  MoveL 1900 to (-42.03, -4.8, 85) mm, rotated rx 180 ry 0 rz -180 deg; joints [35.612, 47.892, 27.55, -143.499, 78.209, -188.599]
  Set speed (130.0 mm/s)
  MoveL 1901 to (-54.1, -7.67, 85) mm, rotated rx 180 ry 0 rz -180 deg; joints [36.421, 46.753, 30.307, -142.872, 79.619, -187.768]
  Call Extruder(18350.601)
  Set speed (30.0 mm/s)
  MoveL 1902 to (-53.59, -12.23, 85) mm, rotated rx 180 ry 0 rz -180 deg; joints [35.732, 46.533, 30.847, -143.601, 79.784, -187.449]
  Call Extruder(18361.531)
  MoveL 1903 to (-49.53, -23.85, 85) mm, rotated rx 180 ry 0 rz -180 deg; joints [33.663, 46.219, 31.622, -145.735, 79.903, -186.811]
  Call Extruder(18372.461)
  MoveL 1904 to (-42.98, -34.27, 85) mm, rotated rx 180 ry 0 rz -180 deg; joints [31.506, 46.21, 31.644, -147.914, 79.666, -186.417]
  Call Extruder(18383.391)
  MoveL 1905 to (-34.27, -42.98, 85) mm, rotated rx 180 ry 0 rz -180 deg; joints [29.427, 46.506, 30.913, -149.974, 79.064, -186.258]
  Call Extruder(18394.322)
  MoveL 1906 to (-23.85, -49.52, 85) mm, rotated rx 180 ry 0 rz 180 deg; joints [27.581, 47.095, 29.473, -151.762, 78.118, -186.31]
  Call Extruder(18405.252)
  MoveL 1907 to (-12.23, -53.59, 85) mm, rotated rx 180 ry 0 rz 180 deg; joints [26.087, 47.95, 27.412, -153.159, 76.881, -186.552]
  Call Extruder(18416.182)
  MoveL 1908 to (0, -54.97, 85) mm, rotated rx 180 ry 0 rz -180 deg; joints [25.019, 49.033, 24.845, -154.089, 75.426, -186.97]
  Call Extruder(18421.833)
  MoveL 1909 to (6.32, -54.26, 85) mm, rotated rx -180 ry 0 rz -180 deg; joints [24.697, 49.678, 23.338, -154.319, 74.609, -187.273]
  Call Extruder(18427.112)
  MoveL 1910 to (12.23, -53.59, 85) mm, rotated rx -180 ry 0 rz -180 deg; joints [24.406, 50.294, 21.91, -154.52, 73.84, -187.555]
  Call Extruder(18438.042)
  MoveL 1911 to (23.85, -49.52, 85) mm, rotated rx 180 ry 0 rz 180 deg; joints [24.239, 51.674, 18.756, -154.459, 72.215, -188.304]
  Call Extruder(18448.973)
  MoveL 1912 to (34.27, -42.98, 85) mm, rotated rx 180 ry 0 rz 180 deg; joints [24.487, 53.106, 15.533, -153.939, 70.641, -189.208]
  Call Extruder(18459.903)
  MoveL 1913 to (42.98, -34.27, 85) mm, rotated rx 180 ry 0 rz 180 deg; joints [25.101, 54.522, 12.393, -153.013, 69.203, -190.249]
  Call Extruder(18470.833)
  MoveL 1914 to (49.52, -23.85, 85) mm, rotated rx 180 ry 0 rz -180 deg; joints [26.025, 55.85, 9.486, -151.751, 67.976, -191.391]
  Call Extruder(18481.763)
  MoveL 1915 to (53.59, -12.23, 85) mm, rotated rx -180 ry 0 rz 180 deg; joints [27.2, 57.019, 6.95, -150.232, 67.025, -192.585]
  Call Extruder(18492.693)
  MoveL 1916 to (54.97, 0, 85) mm, rotated rx -180 ry 0 rz -180 deg; joints [28.57, 57.965, 4.914, -148.541, 66.399, -193.763]
  Call Extruder(18503.624)
  MoveL 1917 to (53.59, 12.23, 85) mm, rotated rx 180 ry 0 rz -180 deg; joints [30.077, 58.634, 3.483, -146.767, 66.128, -194.851]
  Call Extruder(18514.554)
  MoveL 1918 to (49.53, 23.85, 85) mm, rotated rx -180 ry 0 rz -180 deg; joints [31.665, 58.984, 2.736, -144.994, 66.219, -195.771]
  Call Extruder(18525.484)
  MoveL 1919 to (42.98, 34.27, 85) mm, rotated rx 180 ry 0 rz 180 deg; joints [33.282, 58.994, 2.714, -143.296, 66.658, -196.456]
  Call Extruder(18536.414)
  MoveL 1920 to (34.27, 42.98, 85) mm, rotated rx 180 ry 0 rz 180 deg; joints [34.874, 58.664, 3.42, -141.736, 67.412, -196.854]
  Call Extruder(18547.344)
  MoveL 1921 to (23.85, 49.53, 85) mm, rotated rx 180 ry 0 rz 180 deg; joints [36.387, 58.013, 4.812, -140.363, 68.428, -196.939]
  Call Extruder(18558.275)
  MoveL 1922 to (12.23, 53.59, 85) mm, rotated rx 180 ry 0 rz -180 deg; joints [37.766, 57.081, 6.816, -139.215, 69.646, -196.703]
  Call Extruder(18569.205)
  MoveL 1923 to (0, 54.97, 85) mm, rotated rx 180 ry 0 rz 180 deg; joints [38.954, 55.923, 9.325, -138.323, 70.999, -196.165]
  Call Extruder(18580.135)
  MoveL 1924 to (-12.23, 53.59, 85) mm, rotated rx 180 ry 0 rz 180 deg; joints [39.895, 54.603, 12.215, -137.717, 72.421, -195.358]
  Call Extruder(18591.065)
  MoveL 1925 to (-23.85, 49.53, 85) mm, rotated rx 180 ry 0 rz 180 deg; joints [40.528, 53.191, 15.344, -137.428, 73.851, -194.333]
  Call Extruder(18601.995)
  MoveL 1926 to (-34.27, 42.98, 85) mm, rotated rx 180 ry 0 rz -180 deg; joints [40.799, 51.757, 18.566, -137.489, 75.233, -193.151]
  Call Extruder(18612.926)
  MoveL 1927 to (-42.98, 34.27, 85) mm, rotated rx -180 ry 0 rz -180 deg; joints [40.659, 50.372, 21.729, -137.932, 76.518, -191.883]
  Call Extruder(18623.856)
  MoveL 1928 to (-49.53, 23.85, 85) mm, rotated rx 180 ry 0 rz 180 deg; joints [40.072, 49.103, 24.681, -138.778, 77.661, -190.604]
  Call Extruder(18634.786)
  MoveL 1929 to (-53.59, 12.23, 85) mm, rotated rx 180 ry 0 rz 180 deg; joints [39.031, 48.008, 27.273, -140.031, 78.617, -189.393]
  Call Extruder(18645.716)
  MoveL 1930 to (-54.97, 0, 85) mm, rotated rx 180 ry 0 rz 180 deg; joints [37.56, 47.138, 29.368, -141.662, 79.34, -188.322]
  Call Extruder(18651.242)
  MoveL 1931 to (-54.27, -6.18, 85) mm, rotated rx 180 ry 0 rz -180 deg; joints [36.644, 46.826, 30.128, -142.636, 79.565, -187.874]
  Set speed (130.0 mm/s)
  MoveL 1932 to (-49.9, -9.51, 85) mm, rotated rx 180 ry 0 rz 180 deg; joints [35.741, 46.98, 29.754, -143.521, 79.265, -187.842]
  MoveL 1933 to (1.69, -13.14, 85) mm, rotated rx -180 ry 0 rz 180 deg; joints [30.694, 51.344, 19.505, -147.855, 73.614, -190.053]
  Call Extruder(18653.246)
  Set speed (80.0 mm/s)
  MoveL 1934 to (2.97, -12.99, 85) mm, rotated rx 180 ry 0 rz -180 deg; joints [30.614, 51.477, 19.201, -147.91, 73.456, -190.124]
  Call Extruder(18657.910)
  MoveL 1935 to (5.78, -12.01, 85) mm, rotated rx 180 ry 0 rz -180 deg; joints [30.526, 51.813, 18.439, -147.933, 73.079, -190.334]
  Call Extruder(18662.573)
  MoveL 1936 to (8.31, -10.42, 85) mm, rotated rx 180 ry 0 rz -180 deg; joints [30.538, 52.16, 17.656, -147.849, 72.712, -190.58]
  Call Extruder(18667.238)
  MoveL 1937 to (10.42, -8.31, 85) mm, rotated rx -180 ry 0 rz -180 deg; joints [30.649, 52.499, 16.893, -147.664, 72.374, -190.852]
  Call Extruder(18671.901)
  MoveL 1938 to (12.01, -5.78, 85) mm, rotated rx 180 ry 0 rz 180 deg; joints [30.85, 52.813, 16.187, -147.389, 72.082, -191.136]
  Call Extruder(18676.565)
  MoveL 1939 to (12.99, -2.97, 85) mm, rotated rx 180 ry 0 rz 180 deg; joints [31.131, 53.088, 15.574, -147.04, 71.852, -191.418]
  Call Extruder(18681.229)
  MoveL 1940 to (13.33, 0, 85) mm, rotated rx 180 ry 0 rz -180 deg; joints [31.476, 53.308, 15.084, -146.635, 71.695, -191.685]
  Call Extruder(18685.893)
  MoveL 1941 to (13, 2.97, 85) mm, rotated rx 180 ry 0 rz -180 deg; joints [31.869, 53.462, 14.741, -146.195, 71.618, -191.923]
  Call Extruder(18690.556)
  MoveL 1942 to (12.01, 5.78, 85) mm, rotated rx -180 ry 0 rz -180 deg; joints [32.292, 53.542, 14.562, -145.741, 71.624, -192.118]
  Call Extruder(18695.220)
  MoveL 1943 to (10.42, 8.31, 85) mm, rotated rx -180 ry 0 rz 180 deg; joints [32.725, 53.544, 14.557, -145.294, 71.713, -192.26]
  Call Extruder(18699.884)
  MoveL 1944 to (8.31, 10.42, 85) mm, rotated rx 180 ry 0 rz 180 deg; joints [33.149, 53.469, 14.725, -144.876, 71.88, -192.341]
  Call Extruder(18704.548)
  MoveL 1945 to (5.78, 12.01, 85) mm, rotated rx 180 ry 0 rz -180 deg; joints [33.544, 53.319, 15.059, -144.504, 72.114, -192.354]
  Call Extruder(18709.211)
  MoveL 1946 to (2.97, 13, 85) mm, rotated rx 180 ry 0 rz 180 deg; joints [33.893, 53.102, 15.541, -144.196, 72.405, -192.301]
  Call Extruder(18713.875)
  MoveL 1947 to (0, 13.33, 85) mm, rotated rx -180 ry 0 rz -180 deg; joints [34.177, 52.831, 16.148, -143.967, 72.737, -192.182]
  Call Extruder(18718.539)
  MoveL 1948 to (-2.97, 13, 85) mm, rotated rx 180 ry 0 rz -180 deg; joints [34.384, 52.518, 16.85, -143.826, 73.094, -192.004]
  Call Extruder(18723.203)
  MoveL 1949 to (-5.78, 12.01, 85) mm, rotated rx 180 ry 0 rz 180 deg; joints [34.5, 52.18, 17.61, -143.782, 73.459, -191.778]
  Call Extruder(18727.866)
  MoveL 1950 to (-8.31, 10.42, 85) mm, rotated rx -180 ry 0 rz -180 deg; joints [34.518, 51.834, 18.393, -143.839, 73.815, -191.515]
  Call Extruder(18732.531)
  MoveL 1951 to (-10.42, 8.31, 85) mm, rotated rx 180 ry 0 rz -180 deg; joints [34.436, 51.496, 19.158, -143.995, 74.144, -191.229]
  Call Extruder(18737.194)
  MoveL 1952 to (-12.01, 5.78, 85) mm, rotated rx -180 ry 0 rz 180 deg; joints [34.254, 51.185, 19.867, -144.246, 74.431, -190.937]
  Call Extruder(18741.858)
  MoveL 1953 to (-12.99, 2.97, 85) mm, rotated rx 180 ry 0 rz -180 deg; joints [33.981, 50.915, 20.484, -144.58, 74.662, -190.654]
  Call Extruder(18746.522)
  MoveL 1954 to (-13.33, 0, 85) mm, rotated rx -180 ry 0 rz -180 deg; joints [33.63, 50.699, 20.978, -144.982, 74.826, -190.393]
  Call Extruder(18751.186)
  MoveL 1955 to (-13, -2.97, 85) mm, rotated rx 180 ry 0 rz 180 deg; joints [33.218, 50.548, 21.325, -145.432, 74.913, -190.167]
  Call Extruder(18755.849)
  MoveL 1956 to (-12.01, -5.78, 85) mm, rotated rx 180 ry 0 rz 180 deg; joints [32.767, 50.47, 21.505, -145.908, 74.918, -189.988]
  Call Extruder(18760.513)
  MoveL 1957 to (-10.42, -8.31, 85) mm, rotated rx -180 ry 0 rz 180 deg; joints [32.302, 50.467, 21.51, -146.382, 74.841, -189.863]
  Call Extruder(18765.177)
  MoveL 1958 to (-8.31, -10.42, 85) mm, rotated rx 180 ry 0 rz -180 deg; joints [31.85, 50.541, 21.34, -146.829, 74.683, -189.797]
  Call Extruder(18769.841)
  MoveL 1959 to (-5.78, -12.01, 85) mm, rotated rx -180 ry 0 rz 180 deg; joints [31.435, 50.688, 21.003, -147.225, 74.453, -189.791]
  Call Extruder(18774.504)
  MoveL 1960 to (-2.97, -12.99, 85) mm, rotated rx 180 ry 0 rz 180 deg; joints [31.079, 50.9, 20.517, -147.548, 74.161, -189.846]
  Call Extruder(18779.168)
  MoveL 1961 to (0, -13.33, 85) mm, rotated rx 180 ry 0 rz -180 deg; joints [30.801, 51.168, 19.906, -147.78, 73.823, -189.959]
  Call Extruder(18781.828)
  MoveL 1962 to (1.69, -13.14, 85) mm, rotated rx -180 ry 0 rz 180 deg; joints [30.694, 51.344, 19.505, -147.855, 73.614, -190.053]
  Set speed (130.0 mm/s)
  MoveL 1963 to (1.69, -13.14, 90) mm, rotated rx -180 ry 0 rz 180 deg; joints [30.694, 50.443, 19.819, -147.761, 73.118, -190.379]
  MoveL 1964 to (-26.25, -4.54, 90) mm, rotated rx 180 ry 0 rz -180 deg; joints [34.172, 48.315, 24.645, -144.623, 75.968, -189.768]
  Call Extruder(18784.060)
  Set speed (60.0 mm/s)
  MoveL 1965 to (-26.09, -5.96, 90) mm, rotated rx 180 ry 0 rz -180 deg; joints [33.969, 48.243, 24.81, -144.843, 76.01, -189.663]
  Call Extruder(18793.425)
  MoveL 1966 to (-24.12, -11.61, 90) mm, rotated rx 180 ry 0 rz 180 deg; joints [33.033, 48.083, 25.176, -145.823, 76.027, -189.311]
  Call Extruder(18802.790)
  MoveL 1967 to (-20.93, -16.69, 90) mm, rotated rx 180 ry 0 rz -180 deg; joints [32.066, 48.079, 25.187, -146.809, 75.877, -189.069]
  Call Extruder(18812.155)
  MoveL 1968 to (-16.69, -20.93, 90) mm, rotated rx 180 ry 0 rz 180 deg; joints [31.126, 48.229, 24.841, -147.739, 75.565, -188.942]
  Call Extruder(18821.520)
  MoveL 1969 to (-11.61, -24.11, 90) mm, rotated rx 180 ry 0 rz -180 deg; joints [30.272, 48.527, 24.158, -148.558, 75.105, -188.931]
  Call Extruder(18830.885)
  MoveL 1970 to (-5.96, -26.09, 90) mm, rotated rx -180 ry 0 rz -180 deg; joints [29.552, 48.958, 23.173, -149.218, 74.519, -189.035]
  Call Extruder(18840.250)
  MoveL 1971 to (0, -26.77, 90) mm, rotated rx -180 ry 0 rz -180 deg; joints [29.003, 49.501, 21.939, -149.681, 73.837, -189.246]
  Call Extruder(18845.916)
  MoveL 1972 to (3.6, -26.36, 90) mm, rotated rx 180 ry 0 rz 180 deg; joints [28.788, 49.881, 21.082, -149.832, 73.389, -189.435]
  Call Extruder(18849.615)
  MoveL 1973 to (5.96, -26.09, 90) mm, rotated rx 180 ry 0 rz 180 deg; joints [28.65, 50.131, 20.519, -149.926, 73.096, -189.558]
  Call Extruder(18858.980)
  MoveL 1974 to (11.61, -24.11, 90) mm, rotated rx 180 ry 0 rz -180 deg; joints [28.503, 50.816, 18.985, -149.946, 72.336, -189.958]
  Call Extruder(18868.345)
  MoveL 1975 to (16.69, -20.93, 90) mm, rotated rx 180 ry 0 rz -180 deg; joints [28.559, 51.523, 17.413, -149.746, 71.598, -190.433]
  Call Extruder(18877.710)
  MoveL 1976 to (20.93, -16.69, 90) mm, rotated rx 180 ry 0 rz 180 deg; joints [28.808, 52.216, 15.882, -149.344, 70.922, -190.964]
  Call Extruder(18887.075)
  MoveL 1977 to (24.12, -11.61, 90) mm, rotated rx -180 ry 0 rz 180 deg; joints [29.229, 52.861, 14.466, -148.767, 70.343, -191.529]
  Call Extruder(18896.440)
  MoveL 1978 to (26.09, -5.96, 90) mm, rotated rx 180 ry 0 rz 180 deg; joints [29.796, 53.424, 13.236, -148.05, 69.891, -192.102]
  Call Extruder(18905.805)
  MoveL 1979 to (26.77, 0, 90) mm, rotated rx 180 ry 0 rz -180 deg; joints [30.482, 53.877, 12.252, -147.232, 69.589, -192.652]
  Call Extruder(18915.170)
  MoveL 1980 to (26.09, 5.96, 90) mm, rotated rx 180 ry 0 rz -180 deg; joints [31.252, 54.194, 11.564, -146.354, 69.451, -193.15]
  Call Extruder(18924.535)
  MoveL 1981 to (24.11, 11.61, 90) mm, rotated rx -180 ry 0 rz 180 deg; joints [32.076, 54.36, 11.205, -145.458, 69.481, -193.565]
  Call Extruder(18933.900)
  MoveL 1982 to (20.93, 16.69, 90) mm, rotated rx 180 ry 0 rz -180 deg; joints [32.917, 54.365, 11.195, -144.584, 69.676, -193.873]
  Call Extruder(18943.265)
  MoveL 1983 to (16.69, 20.93, 90) mm, rotated rx 180 ry 0 rz -180 deg; joints [33.742, 54.208, 11.533, -143.77, 70.023, -194.053]
  Call Extruder(18952.630)
  MoveL 1984 to (11.61, 24.12, 90) mm, rotated rx -180 ry 0 rz 180 deg; joints [34.517, 53.899, 12.203, -143.049, 70.501, -194.094]
  Call Extruder(18961.995)
  MoveL 1985 to (5.96, 26.09, 90) mm, rotated rx 180 ry 0 rz -180 deg; joints [35.208, 53.454, 13.171, -142.449, 71.085, -193.993]
  Call Extruder(18971.360)
  MoveL 1986 to (0, 26.77, 90) mm, rotated rx 180 ry 0 rz 180 deg; joints [35.784, 52.897, 14.388, -141.996, 71.744, -193.754]
  Call Extruder(18980.725)
  MoveL 1987 to (-5.96, 26.09, 90) mm, rotated rx 180 ry 0 rz 180 deg; joints [36.214, 52.256, 15.795, -141.709, 72.448, -193.392]
  Call Extruder(18990.090)
  MoveL 1988 to (-11.61, 24.12, 90) mm, rotated rx 180 ry 0 rz -180 deg; joints [36.473, 51.564, 17.321, -141.605, 73.162, -192.928]
  Call Extruder(18999.455)
  MoveL 1989 to (-16.69, 20.93, 90) mm, rotated rx 180 ry 0 rz -180 deg; joints [36.542, 50.857, 18.893, -141.694, 73.854, -192.389]
  Call Extruder(19008.820)
  MoveL 1990 to (-20.93, 16.69, 90) mm, rotated rx -180 ry 0 rz 180 deg; joints [36.407, 50.17, 20.431, -141.981, 74.495, -191.805]
  Call Extruder(19018.185)
  MoveL 1991 to (-24.12, 11.61, 90) mm, rotated rx -180 ry 0 rz -180 deg; joints [36.065, 49.536, 21.86, -142.46, 75.056, -191.209]
  Call Extruder(19027.550)
  MoveL 1992 to (-26.09, 5.96, 90) mm, rotated rx 180 ry 0 rz -180 deg; joints [35.528, 48.987, 23.107, -143.116, 75.509, -190.634]
  Call Extruder(19036.915)
  MoveL 1993 to (-26.77, 0, 90) mm, rotated rx 180 ry 0 rz -180 deg; joints [34.817, 48.549, 24.108, -143.924, 75.834, -190.11]
  Call Extruder(19041.703)
  MoveL 1994 to (-26.42, -3.05, 90) mm, rotated rx -180 ry 0 rz -180 deg; joints [34.385, 48.391, 24.47, -144.392, 75.924, -189.88]
  Set speed (130.0 mm/s)
  MoveL 1995 to (-41.86, -6.29, 90) mm, rotated rx 180 ry 0 rz -180 deg; joints [35.393, 46.847, 28.05, -143.651, 77.737, -188.884]
  Call Extruder(19046.701)
  Set speed (60.0 mm/s)
  MoveL 1996 to (-41.5, -9.47, 90) mm, rotated rx 180 ry 0 rz 180 deg; joints [34.924, 46.689, 28.423, -144.152, 77.839, -188.654]
  Call Extruder(19061.597)
  MoveL 1997 to (-38.36, -18.47, 90) mm, rotated rx 180 ry 0 rz -180 deg; joints [33.373, 46.437, 29.016, -145.764, 77.892, -188.124]
  Call Extruder(19076.493)
  MoveL 1998 to (-33.29, -26.54, 90) mm, rotated rx 180 ry 0 rz 180 deg; joints [31.763, 46.43, 29.033, -147.397, 77.677, -187.773]
  Call Extruder(19091.389)
  MoveL 1999 to (-26.54, -33.28, 90) mm, rotated rx 180 ry 0 rz -180 deg; joints [30.206, 46.667, 28.474, -148.94, 77.196, -187.603]
  Call Extruder(19106.284)
  MoveL 2000 to (-18.47, -38.36, 90) mm, rotated rx -180 ry 0 rz 180 deg; joints [28.808, 47.137, 27.372, -150.288, 76.465, -187.607]
  Call Extruder(19121.180)
  MoveL 2001 to (-9.47, -41.5, 90) mm, rotated rx 180 ry 0 rz -180 deg; joints [27.654, 47.818, 25.788, -151.357, 75.523, -187.775]
  Call Extruder(19136.076)
  MoveL 2002 to (0, -42.57, 90) mm, rotated rx -180 ry 0 rz -180 deg; joints [26.805, 48.678, 23.811, -152.086, 74.422, -188.098]
  Call Extruder(19144.508)
  MoveL 2003 to (5.36, -41.97, 90) mm, rotated rx 180 ry 0 rz -180 deg; joints [26.51, 49.239, 22.533, -152.294, 73.745, -188.362]
  Call Extruder(19150.972)
  MoveL 2004 to (9.47, -41.5, 90) mm, rotated rx -180 ry 0 rz -180 deg; joints [26.29, 49.676, 21.543, -152.445, 73.223, -188.565]
  Call Extruder(19165.867)
  MoveL 2005 to (18.47, -38.36, 90) mm, rotated rx -180 ry 0 rz -180 deg; joints [26.114, 50.765, 19.1, -152.431, 71.995, -189.168]
  Call Extruder(19180.763)
  MoveL 2006 to (26.54, -33.28, 90) mm, rotated rx 180 ry 0 rz 180 deg; joints [26.262, 51.89, 16.601, -152.062, 70.804, -189.891]
  Call Extruder(19195.659)
  MoveL 2007 to (33.28, -26.54, 90) mm, rotated rx -180 ry 0 rz -180 deg; joints [26.703, 52.997, 14.168, -151.375, 69.715, -190.715]
  Call Extruder(19210.555)
  MoveL 2008 to (38.36, -18.47, 90) mm, rotated rx 180 ry 0 rz 180 deg; joints [27.4, 54.031, 11.918, -150.419, 68.787, -191.607]
  Call Extruder(19225.451)
  MoveL 2009 to (41.5, -9.47, 90) mm, rotated rx 180 ry 0 rz -180 deg; joints [28.309, 54.937, 9.96, -149.255, 68.067, -192.526]
  Call Extruder(19240.347)
  MoveL 2010 to (42.57, 0, 90) mm, rotated rx 180 ry 0 rz 180 deg; joints [29.382, 55.667, 8.391, -147.947, 67.593, -193.424]
  Call Extruder(19255.242)
  MoveL 2011 to (41.5, 9.47, 90) mm, rotated rx 180 ry 0 rz -180 deg; joints [30.575, 56.181, 7.292, -146.562, 67.386, -194.247]
  Call Extruder(19270.138)
  MoveL 2012 to (38.36, 18.47, 90) mm, rotated rx -180 ry 0 rz 180 deg; joints [31.839, 56.449, 6.719, -145.166, 67.452, -194.941]
  Call Extruder(19285.034)
  MoveL 2013 to (33.28, 26.54, 90) mm, rotated rx 180 ry 0 rz -180 deg; joints [33.128, 56.457, 6.702, -143.819, 67.783, -195.459]
  Call Extruder(19299.930)
  MoveL 2014 to (26.54, 33.29, 90) mm, rotated rx 180 ry 0 rz -180 deg; joints [34.394, 56.204, 7.243, -142.573, 68.354, -195.764]
  Call Extruder(19314.826)
  MoveL 2015 to (18.47, 38.36, 90) mm, rotated rx 180 ry 0 rz -180 deg; joints [35.592, 55.703, 8.313, -141.473, 69.129, -195.837]
  Call Extruder(19329.721)
  MoveL 2016 to (9.47, 41.51, 90) mm, rotated rx 180 ry 0 rz -180 deg; joints [36.675, 54.985, 9.856, -140.555, 70.064, -195.67]
  Call Extruder(19344.617)
  MoveL 2017 to (0, 42.57, 90) mm, rotated rx 180 ry 0 rz -180 deg; joints [37.594, 54.088, 11.794, -139.85, 71.109, -195.277]
  Call Extruder(19359.513)
  MoveL 2018 to (-9.47, 41.51, 90) mm, rotated rx 180 ry 0 rz -180 deg; joints [38.304, 53.061, 14.03, -139.386, 72.213, -194.679]
  Call Extruder(19374.409)
  MoveL 2019 to (-18.47, 38.36, 90) mm, rotated rx 180 ry 0 rz -180 deg; joints [38.762, 51.956, 16.455, -139.189, 73.327, -193.915]
  Call Extruder(19389.304)
  MoveL 2020 to (-26.54, 33.29, 90) mm, rotated rx 180 ry 0 rz -180 deg; joints [38.928, 50.83, 18.953, -139.28, 74.405, -193.029]
  Call Extruder(19404.200)
  MoveL 2021 to (-33.29, 26.54, 90) mm, rotated rx 180 ry 0 rz 180 deg; joints [38.772, 49.738, 21.403, -139.676, 75.404, -192.074]
  Call Extruder(19419.096)
  MoveL 2022 to (-38.36, 18.47, 90) mm, rotated rx 180 ry 0 rz 180 deg; joints [38.277, 48.734, 23.684, -140.383, 76.283, -191.106]
  Call Extruder(19433.992)
  MoveL 2023 to (-41.5, 9.47, 90) mm, rotated rx 180 ry 0 rz -180 deg; joints [37.447, 47.864, 25.682, -141.391, 77.005, -190.18]
  Call Extruder(19448.888)
  MoveL 2024 to (-42.57, 0, 90) mm, rotated rx 180 ry 0 rz 180 deg; joints [36.31, 47.172, 27.291, -142.667, 77.535, -189.349]
  Call Extruder(19456.442)
  MoveL 2025 to (-42.03, -4.8, 90) mm, rotated rx -180 ry 0 rz -180 deg; joints [35.612, 46.923, 27.873, -143.416, 77.689, -188.993]
  Set speed (130.0 mm/s)
  MoveL 2026 to (-54.1, -7.67, 90) mm, rotated rx 180 ry 0 rz -180 deg; joints [36.421, 45.756, 30.634, -142.796, 79.086, -188.18]
  Call Extruder(19460.515)
  Set speed (30.0 mm/s)
  MoveL 2027 to (-53.59, -12.23, 90) mm, rotated rx 180 ry 0 rz 180 deg; joints [35.732, 45.53, 31.175, -143.527, 79.242, -187.857]
  Call Extruder(19471.445)
  MoveL 2028 to (-49.53, -23.85, 90) mm, rotated rx 180 ry 0 rz -180 deg; joints [33.663, 45.208, 31.951, -145.665, 79.34, -187.201]
  Call Extruder(19482.375)
  MoveL 2029 to (-42.98, -34.27, 90) mm, rotated rx -180 ry 0 rz -180 deg; joints [31.506, 45.199, 31.974, -147.846, 79.089, -186.786]
  Call Extruder(19493.305)
  MoveL 2030 to (-34.27, -42.98, 90) mm, rotated rx 180 ry 0 rz -180 deg; joints [29.427, 45.503, 31.241, -149.907, 78.479, -186.602]
  Call Extruder(19504.235)
  MoveL 2031 to (-23.85, -49.52, 90) mm, rotated rx 180 ry 0 rz 180 deg; joints [27.581, 46.107, 29.799, -151.694, 77.535, -186.631]
  Call Extruder(19515.166)
  MoveL 2032 to (-12.23, -53.59, 90) mm, rotated rx 180 ry 0 rz 180 deg; joints [26.087, 46.982, 27.734, -153.089, 76.305, -186.852]
  Call Extruder(19526.096)
  MoveL 2033 to (0, -54.97, 90) mm, rotated rx -180 ry 0 rz -180 deg; joints [25.019, 48.089, 25.164, -154.016, 74.864, -187.252]
  Call Extruder(19532.120)
  MoveL 2034 to (6.74, -54.21, 90) mm, rotated rx -180 ry 0 rz 180 deg; joints [24.676, 48.791, 23.554, -154.259, 74.003, -187.569]
  Call Extruder(19537.026)
  MoveL 2035 to (12.23, -53.59, 90) mm, rotated rx 180 ry 0 rz 180 deg; joints [24.406, 49.374, 22.226, -154.444, 73.296, -187.826]
  Call Extruder(19547.956)
  MoveL 2036 to (23.85, -49.53, 90) mm, rotated rx -180 ry 0 rz -180 deg; joints [24.239, 50.778, 19.069, -154.377, 71.691, -188.568]
  Call Extruder(19558.886)
  MoveL 2037 to (34.27, -42.98, 90) mm, rotated rx -180 ry 0 rz 180 deg; joints [24.487, 52.233, 15.845, -153.851, 70.137, -189.47]
  Call Extruder(19569.817)
  MoveL 2038 to (42.98, -34.27, 90) mm, rotated rx -180 ry 0 rz -180 deg; joints [25.101, 53.668, 12.705, -152.918, 68.72, -190.513]
  Call Extruder(19580.747)
  MoveL 2039 to (49.52, -23.85, 90) mm, rotated rx 180 ry 0 rz -180 deg; joints [26.025, 55.012, 9.798, -151.649, 67.514, -191.66]
  Call Extruder(19591.677)
  MoveL 2040 to (53.59, -12.23, 90) mm, rotated rx 180 ry 0 rz 180 deg; joints [27.2, 56.194, 7.264, -150.123, 66.582, -192.862]
  Call Extruder(19602.607)
  MoveL 2041 to (54.97, 0, 90) mm, rotated rx -180 ry 0 rz -180 deg; joints [28.57, 57.15, 5.229, -148.426, 65.973, -194.049]
  Call Extruder(19613.537)
  MoveL 2042 to (53.59, 12.23, 90) mm, rotated rx 180 ry 0 rz 180 deg; joints [30.077, 57.824, 3.799, -146.646, 65.715, -195.147]
  Call Extruder(19624.468)
  MoveL 2043 to (49.52, 23.85, 90) mm, rotated rx 180 ry 0 rz 180 deg; joints [31.665, 58.178, 3.053, -144.869, 65.818, -196.079]
  Call Extruder(19635.398)
  MoveL 2044 to (42.98, 34.27, 90) mm, rotated rx 180 ry 0 rz -180 deg; joints [33.282, 58.188, 3.031, -143.169, 66.266, -196.775]
  Call Extruder(19646.328)
  MoveL 2045 to (34.27, 42.98, 90) mm, rotated rx 180 ry 0 rz 180 deg; joints [34.874, 57.854, 3.736, -141.608, 67.025, -197.186]
  Call Extruder(19657.258)
  MoveL 2046 to (23.85, 49.53, 90) mm, rotated rx 180 ry 0 rz -180 deg; joints [36.387, 57.198, 5.127, -140.236, 68.043, -197.282]
  Call Extruder(19668.188)
  MoveL 2047 to (12.23, 53.59, 90) mm, rotated rx -180 ry 0 rz 180 deg; joints [37.766, 56.257, 7.129, -139.09, 69.26, -197.06]
  Call Extruder(19679.119)
  MoveL 2048 to (0, 54.97, 90) mm, rotated rx -180 ry 0 rz -180 deg; joints [38.954, 55.086, 9.638, -138.201, 70.608, -196.534]
  Call Extruder(19690.049)
  MoveL 2049 to (-12.23, 53.59, 90) mm, rotated rx 180 ry 0 rz 180 deg; joints [39.895, 53.75, 12.527, -137.6, 72.021, -195.741]
  Call Extruder(19700.979)
  MoveL 2050 to (-23.85, 49.53, 90) mm, rotated rx 180 ry 0 rz -180 deg; joints [40.528, 52.319, 15.656, -137.316, 73.439, -194.728]
  Call Extruder(19711.909)
  MoveL 2051 to (-34.27, 42.98, 90) mm, rotated rx -180 ry 0 rz 180 deg; joints [40.799, 50.863, 18.88, -137.384, 74.805, -193.558]
  Call Extruder(19722.839)
  MoveL 2052 to (-42.98, 34.27, 90) mm, rotated rx 180 ry 0 rz -180 deg; joints [40.659, 49.454, 22.045, -137.833, 76.071, -192.299]
  Call Extruder(19733.770)
  MoveL 2053 to (-49.53, 23.85, 90) mm, rotated rx 180 ry 0 rz 180 deg; joints [40.072, 48.16, 25, -138.686, 77.192, -191.026]
  Call Extruder(19744.700)
  MoveL 2054 to (-53.59, 12.23, 90) mm, rotated rx -180 ry 0 rz -180 deg; joints [39.031, 47.042, 27.595, -139.946, 78.123, -189.816]
  Call Extruder(19755.630)
  MoveL 2055 to (-54.97, 0, 90) mm, rotated rx 180 ry 0 rz -180 deg; joints [37.56, 46.151, 29.693, -141.583, 78.822, -188.741]
  Call Extruder(19761.156)
  MoveL 2056 to (-54.27, -6.18, 90) mm, rotated rx 180 ry 0 rz -180 deg; joints [36.644, 45.831, 30.455, -142.559, 79.034, -188.287]
  Set speed (130.0 mm/s)
  MoveL 2057 to (-49.9, -9.51, 90) mm, rotated rx 180 ry 0 rz -180 deg; joints [35.741, 45.989, 30.08, -143.444, 78.731, -188.245]
  MoveL 2058 to (2.11, -13.09, 90) mm, rotated rx 180 ry 0 rz 180 deg; joints [30.668, 50.487, 19.719, -147.779, 73.066, -190.402]
  Call Extruder(19762.504)
  Set speed (80.0 mm/s)
  MoveL 2059 to (2.97, -12.99, 90) mm, rotated rx 180 ry 0 rz 180 deg; joints [30.614, 50.579, 19.515, -147.816, 72.961, -190.449]
  Call Extruder(19767.168)
  MoveL 2060 to (5.78, -12.01, 90) mm, rotated rx -180 ry 0 rz 180 deg; joints [30.526, 50.92, 18.752, -147.838, 72.588, -190.657]
  Call Extruder(19771.831)
  MoveL 2061 to (8.31, -10.42, 90) mm, rotated rx -180 ry 0 rz 180 deg; joints [30.538, 51.272, 17.969, -147.752, 72.226, -190.901]
  Call Extruder(19776.495)
  MoveL 2062 to (10.42, -8.31, 90) mm, rotated rx 180 ry 0 rz -180 deg; joints [30.649, 51.616, 17.206, -147.565, 71.893, -191.172]
  Call Extruder(19781.159)
  MoveL 2063 to (12.01, -5.78, 90) mm, rotated rx 180 ry 0 rz -180 deg; joints [30.85, 51.936, 16.5, -147.289, 71.606, -191.457]
  Call Extruder(19785.823)
  MoveL 2064 to (12.99, -2.97, 90) mm, rotated rx 180 ry 0 rz -180 deg; joints [31.131, 52.214, 15.886, -146.938, 71.381, -191.74]
  Call Extruder(19790.487)
  MoveL 2065 to (13.33, 0, 90) mm, rotated rx 180 ry 0 rz -180 deg; joints [31.476, 52.437, 15.396, -146.532, 71.229, -192.01]
  Call Extruder(19795.150)
  MoveL 2066 to (12.99, 2.97, 90) mm, rotated rx -180 ry 0 rz -180 deg; joints [31.869, 52.593, 15.053, -146.091, 71.156, -192.25]
  Call Extruder(19799.814)
  MoveL 2067 to (12.01, 5.78, 90) mm, rotated rx 180 ry 0 rz -180 deg; joints [32.292, 52.675, 14.874, -145.636, 71.166, -192.448]
  Call Extruder(19804.478)
  MoveL 2068 to (10.42, 8.31, 90) mm, rotated rx 180 ry 0 rz 180 deg; joints [32.725, 52.677, 14.869, -145.188, 71.258, -192.594]
  Call Extruder(19809.142)
  MoveL 2069 to (8.31, 10.42, 90) mm, rotated rx 180 ry 0 rz 180 deg; joints [33.149, 52.6, 15.038, -144.77, 71.425, -192.678]
  Call Extruder(19813.805)
  MoveL 2070 to (5.78, 12.01, 90) mm, rotated rx 180 ry 0 rz 180 deg; joints [33.544, 52.448, 15.371, -144.398, 71.66, -192.696]
  Call Extruder(19818.469)
  MoveL 2071 to (2.97, 13, 90) mm, rotated rx 180 ry 0 rz 180 deg; joints [33.893, 52.229, 15.854, -144.091, 71.95, -192.646]
  Call Extruder(19823.133)
  MoveL 2072 to (0, 13.33, 90) mm, rotated rx 180 ry 0 rz 180 deg; joints [34.177, 51.953, 16.461, -143.862, 72.28, -192.53]
  Call Extruder(19827.797)
  MoveL 2073 to (-2.97, 13, 90) mm, rotated rx 180 ry 0 rz 180 deg; joints [34.384, 51.636, 17.162, -143.722, 72.635, -192.356]
  Call Extruder(19832.461)
  MoveL 2074 to (-5.78, 12.01, 90) mm, rotated rx 180 ry 0 rz 180 deg; joints [34.5, 51.293, 17.923, -143.68, 72.996, -192.132]
  Call Extruder(19837.124)
  MoveL 2075 to (-8.31, 10.42, 90) mm, rotated rx 180 ry 0 rz 180 deg; joints [34.518, 50.941, 18.706, -143.738, 73.347, -191.871]
  Call Extruder(19841.788)
  MoveL 2076 to (-10.42, 8.31, 90) mm, rotated rx -180 ry 0 rz -180 deg; joints [34.436, 50.598, 19.471, -143.896, 73.672, -191.587]
  Call Extruder(19846.452)
  MoveL 2077 to (-12.01, 5.78, 90) mm, rotated rx 180 ry 0 rz 180 deg; joints [34.254, 50.281, 20.181, -144.148, 73.953, -191.296]
  Call Extruder(19851.116)
  MoveL 2078 to (-12.99, 2.97, 90) mm, rotated rx 180 ry 0 rz 180 deg; joints [33.981, 50.006, 20.799, -144.484, 74.179, -191.011]
  Call Extruder(19855.780)
  MoveL 2079 to (-13.33, 0, 90) mm, rotated rx 180 ry 0 rz 180 deg; joints [33.63, 49.787, 21.294, -144.888, 74.337, -190.748]
  Call Extruder(19860.443)
  MoveL 2080 to (-13, -2.97, 90) mm, rotated rx 180 ry 0 rz -180 deg; joints [33.218, 49.633, 21.64, -145.339, 74.42, -190.521]
  Call Extruder(19865.107)
  MoveL 2081 to (-12.01, -5.78, 90) mm, rotated rx 180 ry 0 rz 180 deg; joints [32.767, 49.554, 21.821, -145.815, 74.421, -190.338]
  Call Extruder(19869.771)
  MoveL 2082 to (-10.42, -8.31, 90) mm, rotated rx -180 ry 0 rz -180 deg; joints [32.302, 49.551, 21.826, -146.29, 74.341, -190.208]
  Call Extruder(19874.435)
  MoveL 2083 to (-8.31, -10.42, 90) mm, rotated rx 180 ry 0 rz 180 deg; joints [31.85, 49.627, 21.656, -146.738, 74.182, -190.137]
  Call Extruder(19879.098)
  MoveL 2084 to (-5.78, -12.01, 90) mm, rotated rx 180 ry 0 rz -180 deg; joints [31.435, 49.776, 21.318, -147.134, 73.951, -190.127]
  Call Extruder(19883.762)
  MoveL 2085 to (-2.97, -12.99, 90) mm, rotated rx 180 ry 0 rz 180 deg; joints [31.079, 49.992, 20.832, -147.456, 73.661, -190.178]
  Call Extruder(19888.426)
  MoveL 2086 to (0, -13.33, 90) mm, rotated rx 180 ry 0 rz 180 deg; joints [30.801, 50.264, 20.22, -147.687, 73.325, -190.287]
  Call Extruder(19891.742)
  MoveL 2087 to (2.11, -13.09, 90) mm, rotated rx 180 ry 0 rz 180 deg; joints [30.668, 50.487, 19.719, -147.779, 73.066, -190.402]
  Set speed (130.0 mm/s)
  MoveL 2088 to (2.11, -13.09, 95) mm, rotated rx 180 ry 0 rz -180 deg; joints [30.668, 49.592, 20.016, -147.681, 72.561, -190.736]
  MoveL 2089 to (-26.25, -4.54, 95) mm, rotated rx 180 ry 0 rz -180 deg; joints [34.172, 47.38, 24.946, -144.529, 75.452, -190.147]
  Call Extruder(19893.974)
  Set speed (60.0 mm/s)
  MoveL 2090 to (-26.09, -5.96, 95) mm, rotated rx 180 ry 0 rz 180 deg; joints [33.969, 47.306, 25.111, -144.75, 75.492, -190.04]
  Call Extruder(19903.339)
  MoveL 2091 to (-24.12, -11.61, 95) mm, rotated rx -180 ry 0 rz 180 deg; joints [33.033, 47.144, 25.478, -145.732, 75.499, -189.681]
  Call Extruder(19912.704)
  MoveL 2092 to (-20.93, -16.69, 95) mm, rotated rx 180 ry 0 rz -180 deg; joints [32.066, 47.139, 25.489, -146.719, 75.344, -189.43]
  Call Extruder(19922.069)
  MoveL 2093 to (-16.69, -20.93, 95) mm, rotated rx 180 ry 0 rz 180 deg; joints [31.126, 47.293, 25.143, -147.65, 75.029, -189.293]
  Call Extruder(19931.434)
  MoveL 2094 to (-11.61, -24.11, 95) mm, rotated rx 180 ry 0 rz 180 deg; joints [30.272, 47.596, 24.459, -148.469, 74.568, -189.272]
  Call Extruder(19940.799)
  MoveL 2095 to (-5.96, -26.09, 95) mm, rotated rx 180 ry 0 rz -180 deg; joints [29.552, 48.036, 23.473, -149.128, 73.984, -189.366]
  Call Extruder(19950.164)
  MoveL 2096 to (0, -26.77, 95) mm, rotated rx 180 ry 0 rz -180 deg; joints [29.003, 48.589, 22.238, -149.59, 73.307, -189.569]
  Call Extruder(19956.486)
  MoveL 2097 to (4.02, -26.31, 95) mm, rotated rx 180 ry 0 rz -180 deg; joints [28.764, 49.02, 21.28, -149.756, 72.813, -189.775]
  Call Extruder(19959.529)
  MoveL 2098 to (5.96, -26.09, 95) mm, rotated rx 180 ry 0 rz 180 deg; joints [28.65, 49.23, 20.816, -149.833, 72.574, -189.874]
  Call Extruder(19968.894)
  MoveL 2099 to (11.61, -24.11, 95) mm, rotated rx 180 ry 0 rz 180 deg; joints [28.503, 49.927, 19.281, -149.85, 71.823, -190.27]
  Call Extruder(19978.259)
  MoveL 2100 to (16.69, -20.93, 95) mm, rotated rx 180 ry 0 rz -180 deg; joints [28.559, 50.645, 17.709, -149.647, 71.095, -190.743]
  Call Extruder(19987.624)
  MoveL 2101 to (20.93, -16.69, 95) mm, rotated rx 180 ry 0 rz 180 deg; joints [28.808, 51.348, 16.177, -149.242, 70.43, -191.274]
  Call Extruder(19996.989)
  MoveL 2102 to (24.12, -11.61, 95) mm, rotated rx 180 ry 0 rz 180 deg; joints [29.229, 52.002, 14.761, -148.661, 69.861, -191.841]
  Call Extruder(20006.354)
  MoveL 2103 to (26.09, -5.96, 95) mm, rotated rx 180 ry 0 rz 180 deg; joints [29.796, 52.573, 13.531, -147.941, 69.42, -192.416]
  Call Extruder(20015.719)
  MoveL 2104 to (26.77, 0, 95) mm, rotated rx 180 ry 0 rz 180 deg; joints [30.482, 53.031, 12.547, -147.119, 69.127, -192.971]
  Call Extruder(20025.084)
  MoveL 2105 to (26.09, 5.96, 95) mm, rotated rx 180 ry 0 rz 180 deg; joints [31.252, 53.353, 11.859, -146.239, 68.996, -193.474]
  Call Extruder(20034.449)
  MoveL 2106 to (24.11, 11.61, 95) mm, rotated rx 180 ry 0 rz -180 deg; joints [32.076, 53.521, 11.5, -145.341, 69.033, -193.896]
  Call Extruder(20043.814)
  MoveL 2107 to (20.93, 16.69, 95) mm, rotated rx 180 ry 0 rz -180 deg; joints [32.917, 53.525, 11.49, -144.466, 69.233, -194.21]
  Call Extruder(20053.179)
  MoveL 2108 to (16.69, 20.93, 95) mm, rotated rx 180 ry 0 rz 180 deg; joints [33.742, 53.367, 11.828, -143.651, 69.583, -194.398]
  Call Extruder(20062.544)
  MoveL 2109 to (11.61, 24.12, 95) mm, rotated rx -180 ry 0 rz -180 deg; joints [34.517, 53.054, 12.498, -142.93, 70.062, -194.446]
  Call Extruder(20071.908)
  MoveL 2110 to (5.96, 26.09, 95) mm, rotated rx -180 ry 0 rz -180 deg; joints [35.208, 52.603, 13.466, -142.332, 70.645, -194.352]
  Call Extruder(20081.274)
  MoveL 2111 to (0, 26.77, 95) mm, rotated rx 180 ry 0 rz 180 deg; joints [35.784, 52.038, 14.683, -141.88, 71.301, -194.12]
  Call Extruder(20090.639)
  MoveL 2112 to (-5.96, 26.09, 95) mm, rotated rx 180 ry 0 rz -180 deg; joints [36.214, 51.388, 16.09, -141.595, 71.999, -193.765]
  Call Extruder(20100.003)
  MoveL 2113 to (-11.61, 24.12, 95) mm, rotated rx 180 ry 0 rz -180 deg; joints [36.473, 50.687, 17.617, -141.494, 72.706, -193.307]
  Call Extruder(20109.368)
  MoveL 2114 to (-16.69, 20.93, 95) mm, rotated rx 180 ry 0 rz -180 deg; joints [36.542, 49.969, 19.189, -141.586, 73.39, -192.772]
  Call Extruder(20118.734)
  MoveL 2115 to (-20.93, 16.69, 95) mm, rotated rx 180 ry 0 rz 180 deg; joints [36.407, 49.27, 20.729, -141.876, 74.021, -192.191]
  Call Extruder(20128.099)
  MoveL 2116 to (-24.12, 11.61, 95) mm, rotated rx 180 ry 0 rz 180 deg; joints [36.065, 48.625, 22.159, -142.358, 74.57, -191.596]
  Call Extruder(20137.463)
  MoveL 2117 to (-26.09, 5.96, 95) mm, rotated rx 180 ry 0 rz 180 deg; joints [35.528, 48.065, 23.407, -143.018, 75.012, -191.02]
  Call Extruder(20146.828)
  MoveL 2118 to (-26.77, 0, 95) mm, rotated rx 180 ry 0 rz -180 deg; joints [34.817, 47.619, 24.409, -143.828, 75.326, -190.493]
  Call Extruder(20151.617)
  MoveL 2119 to (-26.42, -3.05, 95) mm, rotated rx 180 ry 0 rz -180 deg; joints [34.385, 47.458, 24.771, -144.298, 75.411, -190.26]
  Set speed (130.0 mm/s)
  MoveL 2120 to (-41.86, -6.29, 95) mm, rotated rx 180 ry 0 rz 180 deg; joints [35.393, 45.881, 28.356, -143.564, 77.205, -189.285]
  Call Extruder(20156.615)
  Set speed (60.0 mm/s)
  MoveL 2121 to (-41.5, -9.47, 95) mm, rotated rx -180 ry 0 rz 180 deg; joints [34.924, 45.719, 28.73, -144.067, 77.301, -189.052]
  Call Extruder(20171.511)
  MoveL 2122 to (-38.36, -18.47, 95) mm, rotated rx 180 ry 0 rz 180 deg; joints [33.373, 45.462, 29.323, -145.681, 77.339, -188.509]
  Call Extruder(20186.407)
  MoveL 2123 to (-33.28, -26.54, 95) mm, rotated rx 180 ry 0 rz -180 deg; joints [31.763, 45.454, 29.34, -147.316, 77.114, -188.143]
  Call Extruder(20201.302)
  MoveL 2124 to (-26.54, -33.29, 95) mm, rotated rx -180 ry 0 rz -180 deg; joints [30.206, 45.697, 28.78, -148.86, 76.627, -187.955]
  Call Extruder(20216.198)
  MoveL 2125 to (-18.47, -38.36, 95) mm, rotated rx 180 ry 0 rz 180 deg; joints [28.808, 46.178, 27.676, -150.209, 75.897, -187.942]
  Call Extruder(20231.094)
  MoveL 2126 to (-9.47, -41.5, 95) mm, rotated rx -180 ry 0 rz -180 deg; joints [27.654, 46.874, 26.091, -151.276, 74.96, -188.094]
  Call Extruder(20245.990)
  MoveL 2127 to (0, -42.57, 95) mm, rotated rx -180 ry 0 rz -180 deg; joints [26.805, 47.751, 24.111, -152.002, 73.868, -188.403]
  Call Extruder(20255.078)
  MoveL 2128 to (5.78, -41.92, 95) mm, rotated rx 180 ry 0 rz 180 deg; joints [26.488, 48.367, 22.732, -152.224, 73.146, -188.682]
  Call Extruder(20260.886)
  MoveL 2129 to (9.47, -41.5, 95) mm, rotated rx 180 ry 0 rz -180 deg; joints [26.29, 48.768, 21.841, -152.358, 72.682, -188.861]
  Call Extruder(20275.781)
  MoveL 2130 to (18.47, -38.36, 95) mm, rotated rx 180 ry 0 rz 180 deg; joints [26.114, 49.874, 19.396, -152.34, 71.469, -189.458]
  Call Extruder(20290.677)
  MoveL 2131 to (26.54, -33.28, 95) mm, rotated rx 180 ry 0 rz 180 deg; joints [26.262, 51.017, 16.897, -151.966, 70.294, -190.179]
  Call Extruder(20305.573)
  MoveL 2132 to (33.28, -26.54, 95) mm, rotated rx 180 ry 0 rz 180 deg; joints [26.703, 52.14, 14.463, -151.274, 69.223, -191.003]
  Call Extruder(20320.469)
  MoveL 2133 to (38.36, -18.47, 95) mm, rotated rx -180 ry 0 rz -180 deg; joints [27.4, 53.187, 12.213, -150.313, 68.311, -191.898]
  Call Extruder(20335.364)
  MoveL 2134 to (41.51, -9.47, 95) mm, rotated rx 180 ry 0 rz 180 deg; joints [28.309, 54.104, 10.255, -149.143, 67.606, -192.823]
  Call Extruder(20350.260)
  MoveL 2135 to (42.57, 0, 95) mm, rotated rx 180 ry 0 rz 180 deg; joints [29.382, 54.843, 8.687, -147.83, 67.145, -193.729]
  Call Extruder(20365.156)
  MoveL 2136 to (41.51, 9.47, 95) mm, rotated rx 180 ry 0 rz 180 deg; joints [30.575, 55.362, 7.588, -146.441, 66.95, -194.56]
  Call Extruder(20380.052)
  MoveL 2137 to (38.36, 18.47, 95) mm, rotated rx 180 ry 0 rz -180 deg; joints [31.839, 55.634, 7.015, -145.042, 67.026, -195.263]
  Call Extruder(20394.948)
  MoveL 2138 to (33.28, 26.54, 95) mm, rotated rx 180 ry 0 rz 180 deg; joints [33.128, 55.641, 6.999, -143.692, 67.364, -195.791]
  Call Extruder(20409.843)
  MoveL 2139 to (26.54, 33.29, 95) mm, rotated rx 180 ry 0 rz 180 deg; joints [34.394, 55.385, 7.539, -142.446, 67.939, -196.107]
  Call Extruder(20424.739)
  MoveL 2140 to (18.47, 38.36, 95) mm, rotated rx 180 ry 0 rz -180 deg; joints [35.592, 54.88, 8.609, -141.346, 68.716, -196.19]
  Call Extruder(20439.635)
  MoveL 2141 to (9.47, 41.51, 95) mm, rotated rx 180 ry 0 rz 180 deg; joints [36.675, 54.153, 10.151, -140.429, 69.65, -196.034]
  Call Extruder(20454.531)
  MoveL 2142 to (0, 42.57, 95) mm, rotated rx 180 ry 0 rz -180 deg; joints [37.594, 53.245, 12.089, -139.727, 70.69, -195.651]
  Call Extruder(20469.427)
  MoveL 2143 to (-9.47, 41.5, 95) mm, rotated rx -180 ry 0 rz 180 deg; joints [38.304, 52.205, 14.325, -139.267, 71.788, -195.064]
  Call Extruder(20484.322)
  MoveL 2144 to (-18.47, 38.36, 95) mm, rotated rx 180 ry 0 rz 180 deg; joints [38.762, 51.085, 16.751, -139.074, 72.892, -194.309]
  Call Extruder(20499.218)
  MoveL 2145 to (-26.54, 33.29, 95) mm, rotated rx 180 ry 0 rz 180 deg; joints [38.928, 49.941, 19.249, -139.17, 73.956, -193.431]
  Call Extruder(20514.114)
  MoveL 2146 to (-33.29, 26.54, 95) mm, rotated rx 180 ry 0 rz 180 deg; joints [38.772, 48.831, 21.701, -139.571, 74.939, -192.482]
  Call Extruder(20529.010)
  MoveL 2147 to (-38.36, 18.47, 95) mm, rotated rx 180 ry 0 rz 180 deg; joints [38.277, 47.807, 23.984, -140.283, 75.801, -191.517]
  Call Extruder(20543.906)
  MoveL 2148 to (-41.51, 9.47, 95) mm, rotated rx 180 ry 0 rz 180 deg; joints [37.447, 46.921, 25.984, -141.296, 76.504, -190.592]
  Call Extruder(20558.801)
  MoveL 2149 to (-42.57, 0, 95) mm, rotated rx 180 ry 0 rz -180 deg; joints [36.31, 46.213, 27.596, -142.577, 77.015, -189.756]
  Call Extruder(20566.356)
  MoveL 2150 to (-42.03, -4.8, 95) mm, rotated rx 180 ry 0 rz 180 deg; joints [35.612, 45.959, 28.178, -143.329, 77.16, -189.395]
  Set speed (130.0 mm/s)
  MoveL 2151 to (-54.1, -7.67, 95) mm, rotated rx 180 ry 0 rz 180 deg; joints [36.421, 44.764, 30.944, -142.714, 78.542, -188.601]
  Call Extruder(20570.428)
  Set speed (30.0 mm/s)
  MoveL 2152 to (-53.59, -12.23, 95) mm, rotated rx 180 ry 0 rz -180 deg; joints [35.732, 44.532, 31.486, -143.447, 78.689, -188.274]
  Call Extruder(20581.358)
  MoveL 2153 to (-49.53, -23.85, 95) mm, rotated rx -180 ry 0 rz -180 deg; joints [33.663, 44.201, 32.263, -145.589, 78.767, -187.601]
  Call Extruder(20592.289)
  MoveL 2154 to (-42.98, -34.27, 95) mm, rotated rx 180 ry 0 rz -180 deg; joints [31.506, 44.192, 32.286, -147.772, 78.5, -187.163]
  Call Extruder(20603.219)
  MoveL 2155 to (-34.27, -42.98, 95) mm, rotated rx -180 ry 0 rz -180 deg; joints [29.427, 44.504, 31.552, -149.834, 77.884, -186.955]
  Call Extruder(20614.149)
  MoveL 2156 to (-23.85, -49.53, 95) mm, rotated rx 180 ry 0 rz 180 deg; joints [27.581, 45.123, 30.107, -151.622, 76.94, -186.96]
  Call Extruder(20625.079)
  MoveL 2157 to (-12.23, -53.59, 95) mm, rotated rx -180 ry 0 rz -180 deg; joints [26.087, 46.019, 28.039, -153.015, 75.719, -187.159]
  Call Extruder(20636.010)
  MoveL 2158 to (0, -54.97, 95) mm, rotated rx -180 ry 0 rz 180 deg; joints [25.019, 47.15, 25.466, -153.939, 74.291, -187.543]
  Call Extruder(20642.407)
  MoveL 2159 to (7.16, -54.16, 95) mm, rotated rx 180 ry 0 rz 180 deg; joints [24.655, 47.91, 23.754, -154.194, 73.387, -187.871]
  Call Extruder(20646.940)
  MoveL 2160 to (12.23, -53.59, 95) mm, rotated rx 180 ry 0 rz -180 deg; joints [24.406, 48.46, 22.525, -154.363, 72.741, -188.104]
  Call Extruder(20657.870)
  MoveL 2161 to (23.85, -49.53, 95) mm, rotated rx -180 ry 0 rz -180 deg; joints [24.239, 49.888, 19.366, -154.291, 71.156, -188.839]
  Call Extruder(20668.800)
  MoveL 2162 to (34.27, -42.98, 95) mm, rotated rx 180 ry 0 rz -180 deg; joints [24.487, 51.365, 16.14, -153.758, 69.624, -189.739]
  Call Extruder(20679.730)
  MoveL 2163 to (42.98, -34.27, 95) mm, rotated rx -180 ry 0 rz 180 deg; joints [25.101, 52.82, 13, -152.819, 68.228, -190.784]
  Call Extruder(20690.661)
  MoveL 2164 to (49.52, -23.85, 95) mm, rotated rx 180 ry 0 rz -180 deg; joints [26.025, 54.18, 10.094, -151.543, 67.042, -191.937]
  Call Extruder(20701.591)
  MoveL 2165 to (53.59, -12.23, 95) mm, rotated rx -180 ry 0 rz 180 deg; joints [27.2, 55.375, 7.561, -150.009, 66.129, -193.146]
  Call Extruder(20712.521)
  MoveL 2166 to (54.97, 0, 95) mm, rotated rx -180 ry 0 rz 180 deg; joints [28.57, 56.341, 5.527, -148.305, 65.537, -194.343]
  Call Extruder(20723.451)
  MoveL 2167 to (53.59, 12.23, 95) mm, rotated rx -180 ry 0 rz -180 deg; joints [30.077, 57.022, 4.098, -146.52, 65.295, -195.452]
  Call Extruder(20734.381)
  MoveL 2168 to (49.52, 23.85, 95) mm, rotated rx 180 ry 0 rz 180 deg; joints [31.665, 57.379, 3.352, -144.738, 65.409, -196.395]
  Call Extruder(20745.312)
  MoveL 2169 to (42.98, 34.27, 95) mm, rotated rx 180 ry 0 rz -180 deg; joints [33.282, 57.389, 3.331, -143.035, 65.866, -197.103]
  Call Extruder(20756.242)
  MoveL 2170 to (34.27, 42.98, 95) mm, rotated rx 180 ry 0 rz 180 deg; joints [34.874, 57.052, 4.035, -141.474, 66.631, -197.527]
  Call Extruder(20767.172)
  MoveL 2171 to (23.85, 49.53, 95) mm, rotated rx 180 ry 0 rz -180 deg; joints [36.387, 56.389, 5.425, -140.103, 67.651, -197.636]
  Call Extruder(20778.102)
  MoveL 2172 to (12.23, 53.59, 95) mm, rotated rx 180 ry 0 rz -180 deg; joints [37.766, 55.439, 7.426, -138.959, 68.866, -197.426]
  Call Extruder(20789.032)
  MoveL 2173 to (0, 54.97, 95) mm, rotated rx -180 ry 0 rz -180 deg; joints [38.954, 54.256, 9.933, -138.074, 70.209, -196.913]
  Call Extruder(20799.963)
  MoveL 2174 to (-12.23, 53.59, 95) mm, rotated rx 180 ry 0 rz -180 deg; joints [39.895, 52.903, 12.822, -137.477, 71.614, -196.133]
  Call Extruder(20810.893)
  MoveL 2175 to (-23.85, 49.53, 95) mm, rotated rx -180 ry 0 rz -180 deg; joints [40.528, 51.452, 15.952, -137.2, 73.019, -195.133]
  Call Extruder(20821.823)
  MoveL 2176 to (-34.27, 42.98, 95) mm, rotated rx 180 ry 0 rz 180 deg; joints [40.799, 49.974, 19.176, -137.273, 74.37, -193.974]
  Call Extruder(20832.753)
  MoveL 2177 to (-42.98, 34.27, 95) mm, rotated rx -180 ry 0 rz -180 deg; joints [40.659, 48.542, 22.344, -137.729, 75.616, -192.724]
  Call Extruder(20843.683)
  MoveL 2178 to (-49.52, 23.85, 95) mm, rotated rx -180 ry 0 rz -180 deg; joints [40.072, 47.222, 25.302, -138.589, 76.714, -191.458]
  Call Extruder(20854.614)
  MoveL 2179 to (-53.59, 12.23, 95) mm, rotated rx 180 ry 0 rz 180 deg; joints [39.031, 46.08, 27.9, -139.855, 77.621, -190.249]
  Call Extruder(20865.544)
  MoveL 2180 to (-54.97, 0, 95) mm, rotated rx -180 ry 0 rz 180 deg; joints [37.56, 45.168, 30.002, -141.498, 78.294, -189.169]
  Call Extruder(20871.069)
  MoveL 2181 to (-54.27, -6.18, 95) mm, rotated rx 180 ry 0 rz 180 deg; joints [36.644, 44.841, 30.764, -142.476, 78.494, -188.71]
  Set speed (130.0 mm/s)
  MoveL 2182 to (-49.9, -9.51, 95) mm, rotated rx 180 ry 0 rz -180 deg; joints [35.741, 45.002, 30.389, -143.361, 78.187, -188.657]
  MoveL 2183 to (2.53, -13.04, 95) mm, rotated rx 180 ry 0 rz -180 deg; joints [30.642, 49.638, 19.917, -147.699, 72.51, -190.758]
  Call Extruder(20871.762)
  Set speed (80.0 mm/s)
  MoveL 2184 to (2.97, -12.99, 95) mm, rotated rx -180 ry 0 rz 180 deg; joints [30.614, 49.685, 19.812, -147.717, 72.456, -190.782]
  Call Extruder(20876.425)
  MoveL 2185 to (5.78, -12.01, 95) mm, rotated rx -180 ry 0 rz 180 deg; joints [30.526, 50.033, 19.049, -147.737, 72.088, -190.987]
  Call Extruder(20881.089)
  MoveL 2186 to (8.31, -10.42, 95) mm, rotated rx 180 ry 0 rz 180 deg; joints [30.538, 50.39, 18.265, -147.65, 71.73, -191.231]
  Call Extruder(20885.753)
  MoveL 2187 to (10.42, -8.31, 95) mm, rotated rx 180 ry 0 rz -180 deg; joints [30.649, 50.74, 17.502, -147.462, 71.403, -191.501]
  Call Extruder(20890.417)
  MoveL 2188 to (12.01, -5.78, 95) mm, rotated rx -180 ry 0 rz -180 deg; joints [30.85, 51.064, 16.795, -147.184, 71.122, -191.786]
  Call Extruder(20895.080)
  MoveL 2189 to (12.99, -2.97, 95) mm, rotated rx 180 ry 0 rz 180 deg; joints [31.131, 51.346, 16.182, -146.831, 70.902, -192.071]
  Call Extruder(20899.744)
  MoveL 2190 to (13.33, 0, 95) mm, rotated rx 180 ry 0 rz 180 deg; joints [31.476, 51.573, 15.691, -146.424, 70.754, -192.342]
  Call Extruder(20904.408)
  MoveL 2191 to (12.99, 2.97, 95) mm, rotated rx -180 ry 0 rz 180 deg; joints [31.869, 51.731, 15.348, -145.981, 70.685, -192.585]
  Call Extruder(20909.072)
  MoveL 2192 to (12.01, 5.78, 95) mm, rotated rx -180 ry 0 rz -180 deg; joints [32.292, 51.813, 15.169, -145.525, 70.699, -192.787]
  Call Extruder(20913.735)
  MoveL 2193 to (10.42, 8.31, 95) mm, rotated rx 180 ry 0 rz 180 deg; joints [32.725, 51.816, 15.164, -145.077, 70.793, -192.936]
  Call Extruder(20918.400)
  MoveL 2194 to (8.31, 10.42, 95) mm, rotated rx 180 ry 0 rz -180 deg; joints [33.149, 51.738, 15.333, -144.658, 70.962, -193.024]
  Call Extruder(20923.063)
  MoveL 2195 to (5.78, 12.01, 95) mm, rotated rx 180 ry 0 rz -180 deg; joints [33.544, 51.584, 15.667, -144.286, 71.198, -193.046]
  Call Extruder(20927.727)
  MoveL 2196 to (2.97, 13, 95) mm, rotated rx 180 ry 0 rz -180 deg; joints [33.893, 51.361, 16.149, -143.98, 71.487, -193]
  Call Extruder(20932.391)
  MoveL 2197 to (0, 13.33, 95) mm, rotated rx 180 ry 0 rz 180 deg; joints [34.177, 51.082, 16.756, -143.751, 71.816, -192.888]
  Call Extruder(20937.055)
  MoveL 2198 to (-2.97, 13, 95) mm, rotated rx 180 ry 0 rz -180 deg; joints [34.384, 50.76, 17.458, -143.613, 72.167, -192.717]
  Call Extruder(20941.718)
  MoveL 2199 to (-5.78, 12.01, 95) mm, rotated rx 180 ry 0 rz 180 deg; joints [34.5, 50.411, 18.22, -143.572, 72.525, -192.496]
  Call Extruder(20946.382)
  MoveL 2200 to (-8.31, 10.42, 95) mm, rotated rx -180 ry 0 rz 180 deg; joints [34.518, 50.054, 19.003, -143.632, 72.871, -192.237]
  Call Extruder(20951.046)
  MoveL 2201 to (-10.42, 8.31, 95) mm, rotated rx -180 ry 0 rz -180 deg; joints [34.436, 49.705, 19.768, -143.791, 73.19, -191.954]
  Call Extruder(20955.710)
  MoveL 2202 to (-12.01, 5.78, 95) mm, rotated rx 180 ry 0 rz 180 deg; joints [34.254, 49.383, 20.478, -144.045, 73.467, -191.663]
  Call Extruder(20960.373)
  MoveL 2203 to (-12.99, 2.97, 95) mm, rotated rx 180 ry 0 rz 180 deg; joints [33.981, 49.103, 21.097, -144.383, 73.687, -191.377]
  Call Extruder(20965.037)
  MoveL 2204 to (-13.33, 0, 95) mm, rotated rx -180 ry 0 rz 180 deg; joints [33.63, 48.88, 21.592, -144.788, 73.84, -191.113]
  Call Extruder(20969.701)
  MoveL 2205 to (-13, -2.97, 95) mm, rotated rx 180 ry 0 rz -180 deg; joints [33.218, 48.724, 21.939, -145.24, 73.917, -190.882]
  Call Extruder(20974.365)
  MoveL 2206 to (-12.01, -5.78, 95) mm, rotated rx 180 ry 0 rz 180 deg; joints [32.767, 48.643, 22.119, -145.717, 73.915, -190.696]
  Call Extruder(20979.028)
  MoveL 2207 to (-10.42, -8.31, 95) mm, rotated rx 180 ry 0 rz 180 deg; joints [32.302, 48.64, 22.124, -146.193, 73.831, -190.562]
  Call Extruder(20983.693)
  MoveL 2208 to (-8.31, -10.42, 95) mm, rotated rx 180 ry 0 rz 180 deg; joints [31.85, 48.717, 21.954, -146.641, 73.671, -190.487]
  Call Extruder(20988.356)
  MoveL 2209 to (-5.78, -12.01, 95) mm, rotated rx 180 ry 0 rz -180 deg; joints [31.435, 48.869, 21.616, -147.037, 73.44, -190.472]
  Call Extruder(20993.020)
  MoveL 2210 to (-2.97, -13, 95) mm, rotated rx -180 ry 0 rz 180 deg; joints [31.079, 49.089, 21.129, -147.358, 73.15, -190.518]
  Call Extruder(20997.684)
  MoveL 2211 to (0, -13.33, 95) mm, rotated rx -180 ry 0 rz 180 deg; joints [30.801, 49.365, 20.518, -147.589, 72.817, -190.623]
  Call Extruder(21001.655)
  MoveL 2212 to (2.53, -13.04, 95) mm, rotated rx 180 ry 0 rz -180 deg; joints [30.642, 49.638, 19.917, -147.699, 72.51, -190.758]
  Set speed (130.0 mm/s)
  MoveL 2213 to (2.53, -13.04, 100) mm, rotated rx -180 ry 0 rz -180 deg; joints [30.642, 48.749, 20.197, -147.594, 71.996, -191.1]
  MoveL 2214 to (-26.25, -4.54, 100) mm, rotated rx 180 ry 0 rz -180 deg; joints [34.172, 46.45, 25.23, -144.43, 74.927, -190.535]
  Call Extruder(21003.888)
  Set speed (60.0 mm/s)
  MoveL 2215 to (-26.09, -5.96, 100) mm, rotated rx -180 ry 0 rz -180 deg; joints [33.969, 46.376, 25.396, -144.651, 74.964, -190.427]
  Call Extruder(21013.253)
  MoveL 2216 to (-24.12, -11.61, 100) mm, rotated rx 180 ry 0 rz 180 deg; joints [33.033, 46.21, 25.763, -145.636, 74.963, -190.06]
  Call Extruder(21022.618)
  MoveL 2217 to (-20.93, -16.69, 100) mm, rotated rx -180 ry 0 rz 180 deg; joints [32.066, 46.205, 25.773, -146.624, 74.801, -189.799]
  Call Extruder(21031.983)
  MoveL 2218 to (-16.69, -20.93, 100) mm, rotated rx -180 ry 0 rz -180 deg; joints [31.126, 46.361, 25.427, -147.556, 74.482, -189.652]
  Call Extruder(21041.348)
  MoveL 2219 to (-11.61, -24.11, 100) mm, rotated rx 180 ry 0 rz 180 deg; joints [30.272, 46.671, 24.742, -148.375, 74.021, -189.621]
  Call Extruder(21050.713)
  MoveL 2220 to (-5.96, -26.09, 100) mm, rotated rx -180 ry 0 rz 180 deg; joints [29.552, 47.119, 23.756, -149.032, 73.44, -189.706]
  Call Extruder(21060.078)
  MoveL 2221 to (0, -26.77, 100) mm, rotated rx 180 ry 0 rz -180 deg; joints [29.003, 47.683, 22.519, -149.493, 72.769, -189.901]
  Call Extruder(21067.056)
  MoveL 2222 to (4.44, -26.27, 100) mm, rotated rx 180 ry 0 rz 180 deg; joints [28.739, 48.167, 21.461, -149.674, 72.228, -190.123]
  Call Extruder(21069.443)
  MoveL 2223 to (5.96, -26.09, 100) mm, rotated rx 180 ry 0 rz -180 deg; joints [28.65, 48.335, 21.097, -149.734, 72.043, -190.199]
  Call Extruder(21078.808)
  MoveL 2224 to (11.61, -24.12, 100) mm, rotated rx -180 ry 0 rz 180 deg; joints [28.503, 49.043, 19.561, -149.749, 71.301, -190.591]
  Call Extruder(21088.173)
  MoveL 2225 to (16.69, -20.93, 100) mm, rotated rx 180 ry 0 rz 180 deg; joints [28.559, 49.772, 17.988, -149.543, 70.584, -191.061]
  Call Extruder(21097.538)
  MoveL 2226 to (20.93, -16.69, 100) mm, rotated rx 180 ry 0 rz -180 deg; joints [28.808, 50.486, 16.456, -149.134, 69.929, -191.592]
  Call Extruder(21106.903)
  MoveL 2227 to (24.11, -11.61, 100) mm, rotated rx -180 ry 0 rz 180 deg; joints [29.229, 51.15, 15.039, -148.55, 69.371, -192.16]
  Call Extruder(21116.267)
  MoveL 2228 to (26.09, -5.96, 100) mm, rotated rx 180 ry 0 rz -180 deg; joints [29.796, 51.728, 13.809, -147.826, 68.939, -192.739]
  Call Extruder(21125.633)
  MoveL 2229 to (26.77, 0, 100) mm, rotated rx 180 ry 0 rz -180 deg; joints [30.482, 52.192, 12.825, -147.002, 68.656, -193.298]
  Call Extruder(21134.998)
  MoveL 2230 to (26.09, 5.96, 100) mm, rotated rx -180 ry 0 rz -180 deg; joints [31.252, 52.518, 12.137, -146.118, 68.534, -193.807]
  Call Extruder(21144.362)
  MoveL 2231 to (24.11, 11.61, 100) mm, rotated rx 180 ry 0 rz 180 deg; joints [32.076, 52.688, 11.778, -145.218, 68.577, -194.235]
  Call Extruder(21153.727)
  MoveL 2232 to (20.93, 16.69, 100) mm, rotated rx -180 ry 0 rz 180 deg; joints [32.917, 52.693, 11.768, -144.342, 68.782, -194.556]
  Call Extruder(21163.093)
  MoveL 2233 to (16.69, 20.93, 100) mm, rotated rx 180 ry 0 rz 180 deg; joints [33.742, 52.532, 12.106, -143.527, 69.135, -194.751]
  Call Extruder(21172.457)
  MoveL 2234 to (11.61, 24.12, 100) mm, rotated rx 180 ry 0 rz -180 deg; joints [34.517, 52.216, 12.776, -142.806, 69.615, -194.807]
  Call Extruder(21181.822)
  MoveL 2235 to (5.96, 26.09, 100) mm, rotated rx -180 ry 0 rz -180 deg; joints [35.208, 51.759, 13.744, -142.208, 70.197, -194.72]
  Call Extruder(21191.187)
  MoveL 2236 to (0, 26.77, 100) mm, rotated rx 180 ry 0 rz 180 deg; joints [35.784, 51.186, 14.961, -141.758, 70.85, -194.496]
  Call Extruder(21200.552)
  MoveL 2237 to (-5.96, 26.09, 100) mm, rotated rx -180 ry 0 rz -180 deg; joints [36.214, 50.527, 16.368, -141.476, 71.543, -194.147]
  Call Extruder(21209.917)
  MoveL 2238 to (-11.61, 24.12, 100) mm, rotated rx 180 ry 0 rz -180 deg; joints [36.473, 49.815, 17.896, -141.377, 72.242, -193.694]
  Call Extruder(21219.282)
  MoveL 2239 to (-16.69, 20.93, 100) mm, rotated rx 180 ry 0 rz -180 deg; joints [36.542, 49.086, 19.469, -141.473, 72.918, -193.164]
  Call Extruder(21228.647)
  MoveL 2240 to (-20.93, 16.69, 100) mm, rotated rx -180 ry 0 rz 180 deg; joints [36.407, 48.375, 21.009, -141.766, 73.538, -192.586]
  Call Extruder(21238.012)
  MoveL 2241 to (-24.12, 11.61, 100) mm, rotated rx 180 ry 0 rz 180 deg; joints [36.065, 47.719, 22.44, -142.251, 74.076, -191.993]
  Call Extruder(21247.377)
  MoveL 2242 to (-26.09, 5.96, 100) mm, rotated rx 180 ry 0 rz -180 deg; joints [35.528, 47.149, 23.689, -142.914, 74.506, -191.416]
  Call Extruder(21256.742)
  MoveL 2243 to (-26.77, 0, 100) mm, rotated rx 180 ry 0 rz 180 deg; joints [34.817, 46.694, 24.692, -143.727, 74.808, -190.885]
  Call Extruder(21261.531)
  MoveL 2244 to (-26.42, -3.05, 100) mm, rotated rx 180 ry 0 rz 180 deg; joints [34.385, 46.53, 25.055, -144.198, 74.888, -190.649]
  Set speed (130.0 mm/s)
  MoveL 2245 to (-41.86, -6.29, 100) mm, rotated rx 180 ry 0 rz 180 deg; joints [35.393, 44.92, 28.644, -143.471, 76.664, -189.696]
  Call Extruder(21266.529)
  Set speed (60.0 mm/s)
  MoveL 2246 to (-41.5, -9.47, 100) mm, rotated rx -180 ry 0 rz 180 deg; joints [34.924, 44.754, 29.018, -143.975, 76.754, -189.46]
  Call Extruder(21281.424)
  MoveL 2247 to (-38.36, -18.47, 100) mm, rotated rx 180 ry 0 rz 180 deg; joints [33.373, 44.49, 29.612, -145.593, 76.777, -188.904]
  Call Extruder(21296.320)
  MoveL 2248 to (-33.28, -26.54, 100) mm, rotated rx 180 ry 0 rz 180 deg; joints [31.763, 44.483, 29.629, -147.23, 76.541, -188.521]
  Call Extruder(21311.216)
  MoveL 2249 to (-26.54, -33.28, 100) mm, rotated rx 180 ry 0 rz -180 deg; joints [30.206, 44.731, 29.069, -148.775, 76.048, -188.316]
  Call Extruder(21326.112)
  MoveL 2250 to (-18.47, -38.36, 100) mm, rotated rx 180 ry 0 rz -180 deg; joints [28.808, 45.223, 27.964, -150.123, 75.318, -188.285]
  Call Extruder(21341.008)
  MoveL 2251 to (-9.47, -41.5, 100) mm, rotated rx -180 ry 0 rz -180 deg; joints [27.654, 45.934, 26.376, -151.189, 74.386, -188.421]
  Call Extruder(21355.904)
  MoveL 2252 to (0, -42.57, 100) mm, rotated rx 180 ry 0 rz 180 deg; joints [26.805, 46.829, 24.394, -151.914, 73.304, -188.716]
  Call Extruder(21365.647)
  MoveL 2253 to (6.2, -41.87, 100) mm, rotated rx 180 ry 0 rz 180 deg; joints [26.465, 47.503, 22.913, -152.149, 72.539, -189.009]
  Call Extruder(21370.799)
  MoveL 2254 to (9.47, -41.5, 100) mm, rotated rx 180 ry 0 rz 180 deg; joints [26.29, 47.864, 22.122, -152.266, 72.131, -189.164]
  Call Extruder(21385.695)
  MoveL 2255 to (18.47, -38.36, 100) mm, rotated rx 180 ry 0 rz -180 deg; joints [26.114, 48.99, 19.676, -152.244, 70.933, -189.755]
  Call Extruder(21400.591)
  MoveL 2256 to (26.54, -33.28, 100) mm, rotated rx 180 ry 0 rz -180 deg; joints [26.262, 50.151, 17.175, -151.865, 69.775, -190.473]
  Call Extruder(21415.487)
  MoveL 2257 to (33.28, -26.54, 100) mm, rotated rx 180 ry 0 rz -180 deg; joints [26.703, 51.29, 14.741, -151.168, 68.721, -191.298]
  Call Extruder(21430.383)
  MoveL 2258 to (38.36, -18.47, 100) mm, rotated rx 180 ry 0 rz 180 deg; joints [27.4, 52.35, 12.491, -150.201, 67.825, -192.197]
  Call Extruder(21445.278)
  MoveL 2259 to (41.51, -9.47, 100) mm, rotated rx -180 ry 0 rz 180 deg; joints [28.309, 53.278, 10.533, -149.025, 67.136, -193.128]
  Call Extruder(21460.174)
  MoveL 2260 to (42.57, 0, 100) mm, rotated rx 180 ry 0 rz 180 deg; joints [29.382, 54.025, 8.966, -147.707, 66.689, -194.041]
  Call Extruder(21475.070)
  MoveL 2261 to (41.51, 9.47, 100) mm, rotated rx 180 ry 0 rz 180 deg; joints [30.575, 54.55, 7.867, -146.314, 66.506, -194.881]
  Call Extruder(21489.966)
  MoveL 2262 to (38.36, 18.47, 100) mm, rotated rx 180 ry 0 rz -180 deg; joints [31.839, 54.824, 7.294, -144.911, 66.592, -195.594]
  Call Extruder(21504.861)
  MoveL 2263 to (33.28, 26.54, 100) mm, rotated rx 180 ry 0 rz -180 deg; joints [33.128, 54.832, 7.278, -143.56, 66.937, -196.132]
  Call Extruder(21519.757)
  MoveL 2264 to (26.54, 33.28, 100) mm, rotated rx -180 ry 0 rz 180 deg; joints [34.394, 54.574, 7.818, -142.313, 67.518, -196.458]
  Call Extruder(21534.653)
  MoveL 2265 to (18.47, 38.36, 100) mm, rotated rx 180 ry 0 rz 180 deg; joints [35.592, 54.063, 8.887, -141.213, 68.296, -196.552]
  Call Extruder(21549.549)
  MoveL 2266 to (9.47, 41.5, 100) mm, rotated rx 180 ry 0 rz -180 deg; joints [36.675, 53.328, 10.43, -140.298, 69.229, -196.407]
  Call Extruder(21564.445)
  MoveL 2267 to (0, 42.57, 100) mm, rotated rx -180 ry 0 rz -180 deg; joints [37.594, 52.409, 12.366, -139.599, 70.265, -196.034]
  Call Extruder(21579.341)
  MoveL 2268 to (-9.47, 41.51, 100) mm, rotated rx 180 ry 0 rz 180 deg; joints [38.304, 51.355, 14.602, -139.143, 71.355, -195.457]
  Call Extruder(21594.236)
  MoveL 2269 to (-18.47, 38.36, 100) mm, rotated rx 180 ry 0 rz -180 deg; joints [38.762, 50.219, 17.029, -138.954, 72.448, -194.712]
  Call Extruder(21609.132)
  MoveL 2270 to (-26.54, 33.28, 100) mm, rotated rx 180 ry 0 rz 180 deg; joints [38.928, 49.058, 19.529, -139.055, 73.5, -193.843]
  Call Extruder(21624.028)
  MoveL 2271 to (-33.29, 26.54, 100) mm, rotated rx 180 ry 0 rz 180 deg; joints [38.772, 47.929, 21.982, -139.461, 74.467, -192.9]
  Call Extruder(21638.924)
  MoveL 2272 to (-38.36, 18.47, 100) mm, rotated rx 180 ry 0 rz 180 deg; joints [38.277, 46.886, 24.267, -140.178, 75.31, -191.939]
  Call Extruder(21653.819)
  MoveL 2273 to (-41.51, 9.47, 100) mm, rotated rx 180 ry 0 rz 180 deg; joints [37.447, 45.982, 26.27, -141.196, 75.994, -191.013]
  Call Extruder(21668.715)
  MoveL 2274 to (-42.57, 0, 100) mm, rotated rx -180 ry 0 rz -180 deg; joints [36.31, 45.259, 27.883, -142.481, 76.485, -190.173]
  Call Extruder(21676.270)
  MoveL 2275 to (-42.03, -4.8, 100) mm, rotated rx 180 ry 0 rz 180 deg; joints [35.612, 44.999, 28.466, -143.235, 76.622, -189.808]
  Set speed (130.0 mm/s)
  MoveL 2276 to (-54.1, -7.67, 100) mm, rotated rx 180 ry 0 rz -180 deg; joints [36.421, 43.775, 31.236, -142.627, 77.989, -189.032]
  Call Extruder(21680.342)
  Set speed (30.0 mm/s)
  MoveL 2277 to (-53.59, -12.23, 100) mm, rotated rx 180 ry 0 rz 180 deg; joints [35.732, 43.538, 31.779, -143.362, 78.126, -188.7]
  Call Extruder(21691.272)
  MoveL 2278 to (-49.53, -23.85, 100) mm, rotated rx 180 ry 0 rz -180 deg; joints [33.663, 43.199, 32.558, -145.507, 78.183, -188.01]
  Call Extruder(21702.203)
  MoveL 2279 to (-42.98, -34.27, 100) mm, rotated rx 180 ry 0 rz 180 deg; joints [31.506, 43.189, 32.58, -147.693, 77.901, -187.55]
  Call Extruder(21713.133)
  MoveL 2280 to (-34.27, -42.98, 100) mm, rotated rx -180 ry 0 rz 180 deg; joints [29.427, 43.509, 31.845, -149.756, 77.278, -187.317]
  Call Extruder(21724.063)
  MoveL 2281 to (-23.85, -49.52, 100) mm, rotated rx 180 ry 0 rz 180 deg; joints [27.581, 44.144, 30.398, -151.544, 76.335, -187.296]
  Call Extruder(21734.993)
  MoveL 2282 to (-12.23, -53.59, 100) mm, rotated rx 180 ry 0 rz 180 deg; joints [26.087, 45.061, 28.327, -152.936, 75.122, -187.474]
  Call Extruder(21745.923)
  MoveL 2283 to (0, -54.97, 100) mm, rotated rx -180 ry 0 rz 180 deg; joints [25.019, 46.215, 25.75, -153.857, 73.708, -187.84]
  Call Extruder(21752.693)
  MoveL 2284 to (7.58, -54.11, 100) mm, rotated rx 180 ry 0 rz 180 deg; joints [24.634, 47.037, 23.936, -154.124, 72.762, -188.18]
  Call Extruder(21756.854)
  MoveL 2285 to (12.23, -53.59, 100) mm, rotated rx -180 ry 0 rz 180 deg; joints [24.406, 47.551, 22.807, -154.277, 72.175, -188.389]
  Call Extruder(21767.784)
  MoveL 2286 to (23.85, -49.52, 100) mm, rotated rx 180 ry 0 rz -180 deg; joints [24.239, 49.004, 19.645, -154.2, 70.611, -189.117]
  Call Extruder(21778.714)
  MoveL 2287 to (34.27, -42.98, 100) mm, rotated rx -180 ry 0 rz 180 deg; joints [24.487, 50.504, 16.419, -153.661, 69.101, -190.015]
  Call Extruder(21789.644)
  MoveL 2288 to (42.98, -34.27, 100) mm, rotated rx 180 ry 0 rz -180 deg; joints [25.101, 51.979, 13.278, -152.715, 67.727, -191.062]
  Call Extruder(21800.574)
  MoveL 2289 to (49.52, -23.85, 100) mm, rotated rx -180 ry 0 rz 180 deg; joints [26.025, 53.355, 10.372, -151.431, 66.561, -192.221]
  Call Extruder(21811.504)
  MoveL 2290 to (53.59, -12.23, 100) mm, rotated rx 180 ry 0 rz -180 deg; joints [27.2, 54.563, 7.84, -149.89, 65.668, -193.438]
  Call Extruder(21822.435)
  MoveL 2291 to (54.97, 0, 100) mm, rotated rx -180 ry 0 rz -180 deg; joints [28.57, 55.539, 5.807, -148.179, 65.094, -194.646]
  Call Extruder(21833.365)
  MoveL 2292 to (53.59, 12.23, 100) mm, rotated rx 180 ry 0 rz -180 deg; joints [30.077, 56.226, 4.379, -146.388, 64.866, -195.766]
  Call Extruder(21844.295)
  MoveL 2293 to (49.52, 23.85, 100) mm, rotated rx 180 ry 0 rz -180 deg; joints [31.665, 56.586, 3.634, -144.602, 64.993, -196.72]
  Call Extruder(21855.225)
  MoveL 2294 to (42.98, 34.27, 100) mm, rotated rx 180 ry 0 rz -180 deg; joints [33.282, 56.597, 3.612, -142.896, 65.459, -197.441]
  Call Extruder(21866.155)
  MoveL 2295 to (34.27, 42.98, 100) mm, rotated rx -180 ry 0 rz 180 deg; joints [34.874, 56.257, 4.316, -141.334, 66.229, -197.876]
  Call Extruder(21877.086)
  MoveL 2296 to (23.85, 49.53, 100) mm, rotated rx 180 ry 0 rz 180 deg; joints [36.387, 55.588, 5.705, -139.964, 67.252, -197.998]
  Call Extruder(21888.016)
  MoveL 2297 to (12.23, 53.59, 100) mm, rotated rx 180 ry 0 rz 180 deg; joints [37.766, 54.628, 7.705, -138.822, 68.465, -197.801]
  Call Extruder(21898.946)
  MoveL 2298 to (0, 54.97, 100) mm, rotated rx -180 ry 0 rz 180 deg; joints [38.954, 53.432, 10.211, -137.941, 69.803, -197.302]
  Call Extruder(21909.876)
  MoveL 2299 to (-12.23, 53.59, 100) mm, rotated rx 180 ry 0 rz -180 deg; joints [39.895, 52.063, 13.099, -137.349, 71.2, -196.535]
  Call Extruder(21920.806)
  MoveL 2300 to (-23.85, 49.52, 100) mm, rotated rx 180 ry 0 rz -180 deg; joints [40.528, 50.592, 16.23, -137.077, 72.593, -195.548]
  Call Extruder(21931.737)
  MoveL 2301 to (-34.27, 42.98, 100) mm, rotated rx 180 ry 0 rz -180 deg; joints [40.799, 49.092, 19.456, -137.157, 73.927, -194.4]
  Call Extruder(21942.667)
  MoveL 2302 to (-42.98, 34.27, 100) mm, rotated rx 180 ry 0 rz 180 deg; joints [40.659, 47.634, 22.626, -137.619, 75.154, -193.16]
  Call Extruder(21953.597)
  MoveL 2303 to (-49.53, 23.85, 100) mm, rotated rx 180 ry 0 rz -180 deg; joints [40.072, 46.29, 25.586, -138.486, 76.229, -191.899]
  Call Extruder(21964.527)
  MoveL 2304 to (-53.59, 12.23, 100) mm, rotated rx 180 ry 0 rz 180 deg; joints [39.031, 45.123, 28.188, -139.758, 77.11, -190.692]
  Call Extruder(21975.458)
  MoveL 2305 to (-54.97, 0, 100) mm, rotated rx 180 ry 0 rz 180 deg; joints [37.56, 44.19, 30.292, -141.407, 77.756, -189.607]
  Call Extruder(21980.983)
  MoveL 2306 to (-54.27, -6.18, 100) mm, rotated rx 180 ry 0 rz 180 deg; joints [36.644, 43.854, 31.056, -142.388, 77.943, -189.142]
  Set speed (130.0 mm/s)
  MoveL 2307 to (-49.9, -9.51, 100) mm, rotated rx 180 ry 0 rz 180 deg; joints [35.741, 44.02, 30.68, -143.273, 77.632, -189.079]
  MoveL 2308 to (2.94, -13, 100) mm, rotated rx 180 ry 0 rz 180 deg; joints [30.616, 48.795, 20.097, -147.612, 71.946, -191.122]
  Call Extruder(21985.682)
  Set speed (80.0 mm/s)
  MoveL 2309 to (5.78, -12.01, 100) mm, rotated rx 180 ry 0 rz 180 deg; joints [30.526, 49.151, 19.328, -147.632, 71.579, -191.326]
  Call Extruder(21990.346)
  MoveL 2310 to (8.31, -10.42, 100) mm, rotated rx 180 ry 0 rz 180 deg; joints [30.538, 49.514, 18.544, -147.543, 71.226, -191.568]
  Call Extruder(21995.010)
  MoveL 2311 to (10.42, -8.31, 100) mm, rotated rx 180 ry 0 rz 180 deg; joints [30.649, 49.869, 17.78, -147.353, 70.904, -191.838]
  Call Extruder(21999.674)
  MoveL 2312 to (12.01, -5.78, 100) mm, rotated rx 180 ry 0 rz 180 deg; joints [30.85, 50.198, 17.074, -147.073, 70.628, -192.123]
  Call Extruder(22004.337)
  MoveL 2313 to (12.99, -2.97, 100) mm, rotated rx 180 ry 0 rz -180 deg; joints [31.131, 50.484, 16.46, -146.719, 70.414, -192.41]
  Call Extruder(22009.001)
  MoveL 2314 to (13.33, 0, 100) mm, rotated rx 180 ry 0 rz 180 deg; joints [31.476, 50.714, 15.969, -146.31, 70.271, -192.683]
  Call Extruder(22013.665)
  MoveL 2315 to (13, 2.97, 100) mm, rotated rx -180 ry 0 rz 180 deg; joints [31.869, 50.875, 15.626, -145.866, 70.206, -192.929]
  Call Extruder(22018.329)
  MoveL 2316 to (12.01, 5.78, 100) mm, rotated rx 180 ry 0 rz -180 deg; joints [32.292, 50.958, 15.447, -145.409, 70.223, -193.134]
  Call Extruder(22022.992)
  MoveL 2317 to (10.42, 8.31, 100) mm, rotated rx 180 ry 0 rz 180 deg; joints [32.725, 50.961, 15.442, -144.96, 70.32, -193.287]
  Call Extruder(22027.656)
  MoveL 2318 to (8.31, 10.42, 100) mm, rotated rx 180 ry 0 rz 180 deg; joints [33.149, 50.882, 15.611, -144.541, 70.491, -193.379]
  Call Extruder(22032.320)
  MoveL 2319 to (5.78, 12.01, 100) mm, rotated rx -180 ry 0 rz -180 deg; joints [33.544, 50.725, 15.945, -144.169, 70.727, -193.405]
  Call Extruder(22036.984)
  MoveL 2320 to (2.97, 12.99, 100) mm, rotated rx -180 ry 0 rz -180 deg; joints [33.893, 50.5, 16.427, -143.863, 71.016, -193.363]
  Call Extruder(22041.648)
  MoveL 2321 to (0, 13.33, 100) mm, rotated rx -180 ry 0 rz 180 deg; joints [34.177, 50.216, 17.035, -143.636, 71.342, -193.255]
  Call Extruder(22046.312)
  MoveL 2322 to (-2.97, 13, 100) mm, rotated rx 180 ry 0 rz 180 deg; joints [34.384, 49.889, 17.737, -143.498, 71.691, -193.087]
  Call Extruder(22050.975)
  MoveL 2323 to (-5.78, 12.01, 100) mm, rotated rx 180 ry 0 rz 180 deg; joints [34.5, 49.535, 18.499, -143.459, 72.045, -192.869]
  Call Extruder(22055.639)
  MoveL 2324 to (-8.31, 10.42, 100) mm, rotated rx 180 ry 0 rz -180 deg; joints [34.518, 49.172, 19.282, -143.52, 72.387, -192.612]
  Call Extruder(22060.303)
  MoveL 2325 to (-10.42, 8.31, 100) mm, rotated rx -180 ry 0 rz 180 deg; joints [34.436, 48.818, 20.048, -143.681, 72.701, -192.33]
  Call Extruder(22064.967)
  MoveL 2326 to (-12.01, 5.78, 100) mm, rotated rx 180 ry 0 rz 180 deg; joints [34.254, 48.49, 20.759, -143.937, 72.971, -192.039]
  Call Extruder(22069.630)
  MoveL 2327 to (-12.99, 2.97, 100) mm, rotated rx -180 ry 0 rz -180 deg; joints [33.981, 48.206, 21.377, -144.276, 73.186, -191.753]
  Call Extruder(22074.294)
  MoveL 2328 to (-13.33, 0, 100) mm, rotated rx 180 ry 0 rz 180 deg; joints [33.63, 47.979, 21.873, -144.682, 73.333, -191.486]
  Call Extruder(22078.958)
  MoveL 2329 to (-13, -2.97, 100) mm, rotated rx -180 ry 0 rz -180 deg; joints [33.218, 47.82, 22.22, -145.136, 73.406, -191.253]
  Call Extruder(22083.622)
  MoveL 2330 to (-12.01, -5.78, 100) mm, rotated rx 180 ry 0 rz -180 deg; joints [32.767, 47.737, 22.401, -145.614, 73.399, -191.063]
  Call Extruder(22088.285)
  MoveL 2331 to (-10.42, -8.31, 100) mm, rotated rx 180 ry 0 rz -180 deg; joints [32.302, 47.735, 22.406, -146.091, 73.313, -190.925]
  Call Extruder(22092.949)
  MoveL 2332 to (-8.31, -10.42, 100) mm, rotated rx -180 ry 0 rz 180 deg; joints [31.85, 47.813, 22.235, -146.539, 73.151, -190.845]
  Call Extruder(22097.613)
  MoveL 2333 to (-5.78, -12.01, 100) mm, rotated rx 180 ry 0 rz 180 deg; joints [31.435, 47.967, 21.897, -146.935, 72.92, -190.825]
  Call Extruder(22102.277)
  MoveL 2334 to (-2.97, -13, 100) mm, rotated rx -180 ry 0 rz 180 deg; joints [31.079, 48.191, 21.41, -147.256, 72.631, -190.867]
  Call Extruder(22106.941)
  MoveL 2335 to (0, -13.33, 100) mm, rotated rx 180 ry 0 rz 180 deg; joints [30.801, 48.472, 20.798, -147.486, 72.3, -190.968]
  Call Extruder(22111.568)
  MoveL 2336 to (2.94, -13, 100) mm, rotated rx 180 ry 0 rz 180 deg; joints [30.616, 48.795, 20.097, -147.612, 71.946, -191.122]
  Set speed (130.0 mm/s)
  MoveL 2337 to (2.94, -13, 105) mm, rotated rx 180 ry 0 rz -180 deg; joints [30.616, 47.913, 20.36, -147.502, 71.423, -191.472]
  MoveL 2338 to (-26.25, -4.54, 105) mm, rotated rx 180 ry 0 rz -180 deg; joints [34.172, 45.526, 25.497, -144.325, 74.393, -190.932]
  Call Extruder(22113.801)
  Set speed (60.0 mm/s)
  MoveL 2339 to (-26.09, -5.96, 105) mm, rotated rx -180 ry 0 rz -180 deg; joints [33.969, 45.45, 25.663, -144.547, 74.427, -190.822]
  Call Extruder(22123.166)
  MoveL 2340 to (-24.12, -11.61, 105) mm, rotated rx 180 ry 0 rz 180 deg; joints [33.033, 45.281, 26.03, -145.533, 74.417, -190.448]
  Call Extruder(22132.531)
  MoveL 2341 to (-20.93, -16.69, 105) mm, rotated rx 180 ry 0 rz -180 deg; joints [32.066, 45.276, 26.041, -146.523, 74.249, -190.177]
  Call Extruder(22141.896)
  MoveL 2342 to (-16.69, -20.93, 105) mm, rotated rx 180 ry 0 rz 180 deg; joints [31.126, 45.436, 25.694, -147.456, 73.927, -190.02]
  Call Extruder(22151.261)
  MoveL 2343 to (-11.61, -24.12, 105) mm, rotated rx 180 ry 0 rz 180 deg; joints [30.272, 45.751, 25.008, -148.275, 73.465, -189.979]
  Call Extruder(22160.625)
  MoveL 2344 to (-5.96, -26.09, 105) mm, rotated rx 180 ry 0 rz 180 deg; joints [29.552, 46.208, 24.021, -148.932, 72.887, -190.053]
  Call Extruder(22169.991)
  MoveL 2345 to (0, -26.77, 105) mm, rotated rx 180 ry 0 rz -180 deg; joints [29.003, 46.782, 22.784, -149.391, 72.221, -190.24]
  Call Extruder(22177.625)
  MoveL 2346 to (4.86, -26.22, 105) mm, rotated rx 180 ry 0 rz 180 deg; joints [28.715, 47.322, 21.625, -149.587, 71.636, -190.478]
  Call Extruder(22179.356)
  MoveL 2347 to (5.96, -26.09, 105) mm, rotated rx 180 ry 0 rz -180 deg; joints [28.65, 47.445, 21.36, -149.63, 71.502, -190.532]
  Call Extruder(22188.720)
  MoveL 2348 to (11.61, -24.11, 105) mm, rotated rx 180 ry 0 rz 180 deg; joints [28.503, 48.165, 19.823, -149.642, 70.77, -190.919]
  Call Extruder(22198.085)
  MoveL 2349 to (16.69, -20.93, 105) mm, rotated rx 180 ry 0 rz 180 deg; joints [28.559, 48.906, 18.25, -149.433, 70.063, -191.387]
  Call Extruder(22207.451)
  MoveL 2350 to (20.93, -16.69, 105) mm, rotated rx 180 ry 0 rz -180 deg; joints [28.808, 49.631, 16.717, -149.021, 69.419, -191.917]
  Call Extruder(22216.816)
  MoveL 2351 to (24.12, -11.61, 105) mm, rotated rx 180 ry 0 rz 180 deg; joints [29.229, 50.303, 15.3, -148.433, 68.872, -192.487]
  Call Extruder(22226.180)
  MoveL 2352 to (26.09, -5.96, 105) mm, rotated rx 180 ry 0 rz -180 deg; joints [29.796, 50.89, 14.07, -147.706, 68.451, -193.069]
  Call Extruder(22235.545)
  MoveL 2353 to (26.77, 0, 105) mm, rotated rx -180 ry 0 rz 180 deg; joints [30.482, 51.36, 13.086, -146.878, 68.176, -193.633]
  Call Extruder(22244.911)
  MoveL 2354 to (26.09, 5.96, 105) mm, rotated rx 180 ry 0 rz -180 deg; joints [31.252, 51.69, 12.397, -145.992, 68.063, -194.148]
  Call Extruder(22254.275)
  MoveL 2355 to (24.11, 11.61, 105) mm, rotated rx 180 ry 0 rz -180 deg; joints [32.076, 51.861, 12.039, -145.09, 68.113, -194.582]
  Call Extruder(22263.640)
  MoveL 2356 to (20.93, 16.69, 105) mm, rotated rx -180 ry 0 rz -180 deg; joints [32.917, 51.866, 12.029, -144.212, 68.323, -194.911]
  Call Extruder(22273.005)
  MoveL 2357 to (16.69, 20.93, 105) mm, rotated rx -180 ry 0 rz 180 deg; joints [33.742, 51.704, 12.367, -143.397, 68.679, -195.113]
  Call Extruder(22282.370)
  MoveL 2358 to (11.61, 24.12, 105) mm, rotated rx 180 ry 0 rz -180 deg; joints [34.517, 51.383, 13.037, -142.676, 69.16, -195.176]
  Call Extruder(22291.735)
  MoveL 2359 to (5.96, 26.09, 105) mm, rotated rx -180 ry 0 rz -180 deg; joints [35.208, 50.921, 14.004, -142.079, 69.741, -195.097]
  Call Extruder(22301.100)
  MoveL 2360 to (0, 26.77, 105) mm, rotated rx 180 ry 0 rz 180 deg; joints [35.784, 50.341, 15.222, -141.63, 70.391, -194.88]
  Call Extruder(22310.465)
  MoveL 2361 to (-5.96, 26.09, 105) mm, rotated rx 180 ry 0 rz 180 deg; joints [36.214, 49.672, 16.63, -141.351, 71.078, -194.538]
  Call Extruder(22319.830)
  MoveL 2362 to (-11.61, 24.12, 105) mm, rotated rx 180 ry 0 rz -180 deg; joints [36.473, 48.95, 18.157, -141.255, 71.771, -194.091]
  Call Extruder(22329.195)
  MoveL 2363 to (-16.69, 20.93, 105) mm, rotated rx -180 ry 0 rz 180 deg; joints [36.542, 48.209, 19.731, -141.353, 72.437, -193.566]
  Call Extruder(22338.560)
  MoveL 2364 to (-20.93, 16.69, 105) mm, rotated rx 180 ry 0 rz 180 deg; joints [36.407, 47.487, 21.272, -141.649, 73.047, -192.991]
  Call Extruder(22347.925)
  MoveL 2365 to (-24.12, 11.61, 105) mm, rotated rx 180 ry 0 rz -180 deg; joints [36.065, 46.819, 22.704, -142.138, 73.574, -192.399]
  Call Extruder(22357.290)
  MoveL 2366 to (-26.09, 5.96, 105) mm, rotated rx 180 ry 0 rz -180 deg; joints [35.528, 46.239, 23.954, -142.804, 73.992, -191.821]
  Call Extruder(22366.655)
  MoveL 2367 to (-26.77, 0, 105) mm, rotated rx 180 ry 0 rz 180 deg; joints [34.817, 45.775, 24.958, -143.62, 74.282, -191.287]
  Call Extruder(22371.444)
  MoveL 2368 to (-26.42, -3.05, 105) mm, rotated rx 180 ry 0 rz -180 deg; joints [34.385, 45.607, 25.321, -144.093, 74.356, -191.048]
  Set speed (130.0 mm/s)
  MoveL 2369 to (-41.86, -6.29, 105) mm, rotated rx 180 ry 0 rz -180 deg; joints [35.393, 43.963, 28.915, -143.372, 76.114, -190.116]
  Call Extruder(22376.442)
  Set speed (60.0 mm/s)
  MoveL 2370 to (-41.51, -9.47, 105) mm, rotated rx 180 ry 0 rz 180 deg; joints [34.924, 43.793, 29.29, -143.878, 76.197, -189.877]
  Call Extruder(22391.337)
  MoveL 2371 to (-38.36, -18.47, 105) mm, rotated rx 180 ry 0 rz 180 deg; joints [33.373, 43.524, 29.884, -145.498, 76.205, -189.308]
  Call Extruder(22406.233)
  MoveL 2372 to (-33.28, -26.54, 105) mm, rotated rx -180 ry 0 rz -180 deg; joints [31.763, 43.517, 29.902, -147.138, 75.957, -188.908]
  Call Extruder(22421.129)
  MoveL 2373 to (-26.54, -33.28, 105) mm, rotated rx 180 ry 0 rz -180 deg; joints [30.206, 43.771, 29.34, -148.684, 75.459, -188.685]
  Call Extruder(22436.025)
  MoveL 2374 to (-18.47, -38.36, 105) mm, rotated rx -180 ry 0 rz -180 deg; joints [28.808, 44.273, 28.234, -150.033, 74.729, -188.636]
  Call Extruder(22450.920)
  MoveL 2375 to (-9.47, -41.5, 105) mm, rotated rx 180 ry 0 rz -180 deg; joints [27.654, 44.999, 26.644, -151.098, 73.802, -188.755]
  Call Extruder(22465.816)
  MoveL 2376 to (0, -42.57, 105) mm, rotated rx 180 ry 0 rz -180 deg; joints [26.805, 45.912, 24.66, -151.82, 72.73, -189.037]
  Call Extruder(22476.216)
  MoveL 2377 to (6.61, -41.83, 105) mm, rotated rx -180 ry 0 rz -180 deg; joints [26.443, 46.645, 23.078, -152.068, 71.922, -189.343]
  Call Extruder(22480.712)
  MoveL 2378 to (9.47, -41.5, 105) mm, rotated rx 180 ry 0 rz 180 deg; joints [26.29, 46.967, 22.386, -152.17, 71.571, -189.475]
  Call Extruder(22495.608)
  MoveL 2379 to (18.47, -38.36, 105) mm, rotated rx 180 ry 0 rz 180 deg; joints [26.114, 48.111, 19.938, -152.143, 70.388, -190.059]
  Call Extruder(22510.504)
  MoveL 2380 to (26.54, -33.28, 105) mm, rotated rx -180 ry 0 rz 180 deg; joints [26.262, 49.29, 17.436, -151.76, 69.247, -190.775]
  Call Extruder(22525.400)
  MoveL 2381 to (33.28, -26.54, 105) mm, rotated rx -180 ry 0 rz 180 deg; joints [26.703, 50.445, 15.002, -151.056, 68.21, -191.601]
  Call Extruder(22540.295)
  MoveL 2382 to (38.36, -18.47, 105) mm, rotated rx 180 ry 0 rz 180 deg; joints [27.4, 51.52, 12.751, -150.084, 67.331, -192.504]
  Call Extruder(22555.191)
  MoveL 2383 to (41.5, -9.47, 105) mm, rotated rx -180 ry 0 rz -180 deg; joints [28.309, 52.459, 10.794, -148.903, 66.658, -193.441]
  Call Extruder(22570.087)
  MoveL 2384 to (42.57, 0, 105) mm, rotated rx 180 ry 0 rz 180 deg; joints [29.382, 53.214, 9.227, -147.579, 66.225, -194.362]
  Call Extruder(22584.983)
  MoveL 2385 to (41.5, 9.47, 105) mm, rotated rx -180 ry 0 rz -180 deg; joints [30.575, 53.745, 8.129, -146.181, 66.054, -195.211]
  Call Extruder(22599.878)
  MoveL 2386 to (38.36, 18.47, 105) mm, rotated rx -180 ry 0 rz 180 deg; joints [31.839, 54.022, 7.556, -144.775, 66.15, -195.934]
  Call Extruder(22614.774)
  MoveL 2387 to (33.28, 26.54, 105) mm, rotated rx 180 ry 0 rz 180 deg; joints [33.128, 54.03, 7.54, -143.422, 66.503, -196.482]
  Call Extruder(22629.670)
  MoveL 2388 to (26.54, 33.29, 105) mm, rotated rx 180 ry 0 rz -180 deg; joints [34.394, 53.769, 8.08, -142.174, 67.088, -196.819]
  Call Extruder(22644.566)
  MoveL 2389 to (18.47, 38.36, 105) mm, rotated rx 180 ry 0 rz 180 deg; joints [35.592, 53.252, 9.149, -141.075, 67.869, -196.923]
  Call Extruder(22659.462)
  MoveL 2390 to (9.47, 41.51, 105) mm, rotated rx 180 ry 0 rz -180 deg; joints [36.675, 52.509, 10.691, -140.162, 68.8, -196.789]
  Call Extruder(22674.358)
  MoveL 2391 to (0, 42.57, 105) mm, rotated rx -180 ry 0 rz -180 deg; joints [37.594, 51.579, 12.627, -139.465, 69.832, -196.427]
  Call Extruder(22689.253)
  MoveL 2392 to (-9.47, 41.5, 105) mm, rotated rx 180 ry 0 rz -180 deg; joints [38.304, 50.511, 14.863, -139.013, 70.914, -195.861]
  Call Extruder(22704.149)
  MoveL 2393 to (-18.47, 38.36, 105) mm, rotated rx 180 ry 0 rz -180 deg; joints [38.762, 49.359, 17.29, -138.828, 71.998, -195.125]
  Call Extruder(22719.045)
  MoveL 2394 to (-26.54, 33.29, 105) mm, rotated rx 180 ry 0 rz -180 deg; joints [38.928, 48.18, 19.791, -138.934, 73.036, -194.264]
  Call Extruder(22733.941)
  MoveL 2395 to (-33.29, 26.54, 105) mm, rotated rx -180 ry 0 rz -180 deg; joints [38.772, 47.032, 22.246, -139.345, 73.987, -193.328]
  Call Extruder(22748.837)
  MoveL 2396 to (-38.36, 18.47, 105) mm, rotated rx 180 ry 0 rz 180 deg; joints [38.277, 45.971, 24.533, -140.067, 74.812, -192.37]
  Call Extruder(22763.732)
  MoveL 2397 to (-41.5, 9.47, 105) mm, rotated rx 180 ry 0 rz -180 deg; joints [37.447, 45.048, 26.537, -141.09, 75.476, -191.444]
  Call Extruder(22778.628)
  MoveL 2398 to (-42.57, 0, 105) mm, rotated rx 180 ry 0 rz -180 deg; joints [36.31, 44.31, 28.153, -142.38, 75.947, -190.599]
  Call Extruder(22786.182)
  MoveL 2399 to (-42.03, -4.8, 105) mm, rotated rx -180 ry 0 rz 180 deg; joints [35.612, 44.044, 28.737, -143.136, 76.074, -190.23]
  Set speed (130.0 mm/s)
  MoveL 2400 to (-54.1, -7.67, 105) mm, rotated rx 180 ry 0 rz -180 deg; joints [36.421, 42.792, 31.511, -142.533, 77.426, -189.473]
  Call Extruder(22790.255)
  Set speed (30.0 mm/s)
  MoveL 2401 to (-53.59, -12.23, 105) mm, rotated rx 180 ry 0 rz -180 deg; joints [35.732, 42.549, 32.054, -143.27, 77.554, -189.136]
  Call Extruder(22801.185)
  MoveL 2402 to (-49.52, -23.85, 105) mm, rotated rx 180 ry 0 rz -180 deg; joints [33.663, 42.201, 32.834, -145.419, 77.589, -188.428]
  Call Extruder(22812.115)
  MoveL 2403 to (-42.98, -34.27, 105) mm, rotated rx 180 ry 0 rz -180 deg; joints [31.506, 42.191, 32.857, -147.608, 77.292, -187.945]
  Call Extruder(22823.046)
  MoveL 2404 to (-34.27, -42.98, 105) mm, rotated rx 180 ry 0 rz 180 deg; joints [29.427, 42.519, 32.12, -149.673, 76.661, -187.686]
  Call Extruder(22833.976)
  MoveL 2405 to (-23.85, -49.52, 105) mm, rotated rx 180 ry 0 rz -180 deg; joints [27.581, 43.169, 30.671, -151.461, 75.719, -187.641]
  Call Extruder(22844.906)
  MoveL 2406 to (-12.23, -53.59, 105) mm, rotated rx -180 ry 0 rz -180 deg; joints [26.087, 44.108, 28.597, -152.852, 74.514, -187.796]
  Call Extruder(22855.836)
  MoveL 2407 to (0, -54.97, 105) mm, rotated rx 180 ry 0 rz 180 deg; joints [25.019, 45.287, 26.018, -153.77, 73.114, -188.144]
  Call Extruder(22862.979)
  MoveL 2408 to (7.99, -54.07, 105) mm, rotated rx -180 ry 0 rz 180 deg; joints [24.614, 46.171, 24.101, -154.048, 72.128, -188.495]
  Call Extruder(22866.766)
  MoveL 2409 to (12.23, -53.59, 105) mm, rotated rx 180 ry 0 rz -180 deg; joints [24.406, 46.648, 23.071, -154.186, 71.6, -188.681]
  Call Extruder(22877.697)
  MoveL 2410 to (23.85, -49.52, 105) mm, rotated rx 180 ry 0 rz -180 deg; joints [24.239, 48.126, 19.908, -154.104, 70.057, -189.402]
  Call Extruder(22888.627)
  MoveL 2411 to (34.27, -42.98, 105) mm, rotated rx 180 ry 0 rz -180 deg; joints [24.487, 49.648, 16.68, -153.559, 68.569, -190.299]
  Call Extruder(22899.557)
  MoveL 2412 to (42.98, -34.27, 105) mm, rotated rx 180 ry 0 rz 180 deg; joints [25.101, 51.143, 13.539, -152.605, 67.216, -191.348]
  Call Extruder(22910.487)
  MoveL 2413 to (49.53, -23.85, 105) mm, rotated rx 180 ry 0 rz -180 deg; joints [26.025, 52.537, 10.633, -151.314, 66.072, -192.513]
  Call Extruder(22921.417)
  MoveL 2414 to (53.59, -12.23, 105) mm, rotated rx 180 ry 0 rz -180 deg; joints [27.2, 53.758, 8.101, -149.765, 65.199, -193.738]
  Call Extruder(22932.348)
  MoveL 2415 to (54.97, 0, 105) mm, rotated rx -180 ry 0 rz -180 deg; joints [28.57, 54.744, 6.069, -148.047, 64.642, -194.956]
  Call Extruder(22943.278)
  MoveL 2416 to (53.59, 12.23, 105) mm, rotated rx -180 ry 0 rz -180 deg; joints [30.077, 55.438, 4.643, -146.25, 64.429, -196.088]
  Call Extruder(22954.208)
  MoveL 2417 to (49.52, 23.85, 105) mm, rotated rx 180 ry 0 rz 180 deg; joints [31.665, 55.801, 3.898, -144.459, 64.569, -197.054]
  Call Extruder(22965.138)
  MoveL 2418 to (42.98, 34.27, 105) mm, rotated rx 180 ry 0 rz 180 deg; joints [33.282, 55.811, 3.877, -142.751, 65.044, -197.787]
  Call Extruder(22976.068)
  MoveL 2419 to (34.27, 42.98, 105) mm, rotated rx 180 ry 0 rz -180 deg; joints [34.874, 55.469, 4.579, -141.188, 65.82, -198.236]
  Call Extruder(22986.999)
  MoveL 2420 to (23.85, 49.53, 105) mm, rotated rx 180 ry 0 rz -180 deg; joints [36.387, 54.793, 5.968, -139.818, 66.845, -198.37]
  Call Extruder(22997.929)
  MoveL 2421 to (12.23, 53.59, 105) mm, rotated rx 180 ry 0 rz 180 deg; joints [37.766, 53.824, 7.967, -138.68, 68.057, -198.186]
  Call Extruder(23008.859)
  MoveL 2422 to (0, 54.97, 105) mm, rotated rx -180 ry 0 rz 180 deg; joints [38.954, 52.614, 10.472, -137.802, 69.39, -197.7]
  Call Extruder(23019.789)
  MoveL 2423 to (-12.23, 53.59, 105) mm, rotated rx 180 ry 0 rz -180 deg; joints [39.895, 51.229, 13.36, -137.215, 70.778, -196.946]
  Call Extruder(23030.719)
  MoveL 2424 to (-23.85, 49.52, 105) mm, rotated rx 180 ry 0 rz -180 deg; joints [40.528, 49.738, 16.491, -136.949, 72.159, -195.972]
  Call Extruder(23041.650)
  MoveL 2425 to (-34.27, 42.98, 105) mm, rotated rx -180 ry 0 rz 180 deg; joints [40.799, 48.215, 19.718, -137.035, 73.477, -194.836]
  Call Extruder(23052.580)
  MoveL 2426 to (-42.98, 34.27, 105) mm, rotated rx 180 ry 0 rz -180 deg; joints [40.659, 46.732, 22.89, -137.504, 74.684, -193.605]
  Call Extruder(23063.510)
  MoveL 2427 to (-49.53, 23.85, 105) mm, rotated rx 180 ry 0 rz 180 deg; joints [40.072, 45.362, 25.853, -138.376, 75.735, -192.35]
  Call Extruder(23074.440)
  MoveL 2428 to (-53.59, 12.23, 105) mm, rotated rx -180 ry 0 rz 180 deg; joints [39.031, 44.171, 28.458, -139.655, 76.59, -191.144]
  Call Extruder(23085.370)
  MoveL 2429 to (-54.97, 0, 105) mm, rotated rx 180 ry 0 rz 180 deg; joints [37.56, 43.217, 30.565, -141.31, 77.209, -190.054]
  Call Extruder(23090.896)
  MoveL 2430 to (-54.27, -6.18, 105) mm, rotated rx -180 ry 0 rz 180 deg; joints [36.644, 42.873, 31.33, -142.294, 77.384, -189.584]
  Set speed (130.0 mm/s)
  MoveL 2431 to (-49.9, -9.51, 105) mm, rotated rx 180 ry 0 rz -180 deg; joints [35.741, 43.042, 30.954, -143.178, 77.069, -189.511]
  MoveL 2432 to (2.97, -12.99, 105) mm, rotated rx 180 ry 0 rz -180 deg; joints [30.614, 47.916, 20.355, -147.503, 71.421, -191.473]
  Call Extruder(23095.560)
  Set speed (80.0 mm/s)
  MoveL 2433 to (5.78, -12.01, 105) mm, rotated rx 180 ry 0 rz 180 deg; joints [30.526, 48.275, 19.59, -147.52, 71.061, -191.674]
  Call Extruder(23100.223)
  MoveL 2434 to (8.31, -10.42, 105) mm, rotated rx -180 ry 0 rz -180 deg; joints [30.538, 48.644, 18.806, -147.43, 70.713, -191.914]
  Call Extruder(23104.887)
  MoveL 2435 to (10.42, -8.31, 105) mm, rotated rx 180 ry 0 rz 180 deg; joints [30.649, 49.004, 18.042, -147.238, 70.396, -192.183]
  Call Extruder(23109.551)
  MoveL 2436 to (12.01, -5.78, 105) mm, rotated rx -180 ry 0 rz -180 deg; joints [30.85, 49.338, 17.335, -146.957, 70.126, -192.469]
  Call Extruder(23114.215)
  MoveL 2437 to (13, -2.97, 105) mm, rotated rx -180 ry 0 rz -180 deg; joints [31.131, 49.629, 16.721, -146.601, 69.917, -192.757]
  Call Extruder(23118.879)
  MoveL 2438 to (13.33, 0, 105) mm, rotated rx 180 ry 0 rz -180 deg; joints [31.476, 49.862, 16.23, -146.191, 69.779, -193.033]
  Call Extruder(23123.542)
  MoveL 2439 to (12.99, 2.97, 105) mm, rotated rx -180 ry 0 rz 180 deg; joints [31.869, 50.025, 15.887, -145.745, 69.719, -193.281]
  Call Extruder(23128.206)
  MoveL 2440 to (12.01, 5.78, 105) mm, rotated rx 180 ry 0 rz -180 deg; joints [32.292, 50.109, 15.708, -145.287, 69.74, -193.49]
  Call Extruder(23132.870)
  MoveL 2441 to (10.42, 8.31, 105) mm, rotated rx 180 ry 0 rz 180 deg; joints [32.725, 50.112, 15.703, -144.838, 69.839, -193.647]
  Call Extruder(23137.534)
  MoveL 2442 to (8.31, 10.42, 105) mm, rotated rx 180 ry 0 rz -180 deg; joints [33.149, 50.032, 15.872, -144.418, 70.012, -193.743]
  Call Extruder(23142.198)
  MoveL 2443 to (5.78, 12.01, 105) mm, rotated rx 180 ry 0 rz -180 deg; joints [33.544, 49.873, 16.206, -144.047, 70.248, -193.772]
  Call Extruder(23146.861)
  MoveL 2444 to (2.97, 13, 105) mm, rotated rx -180 ry 0 rz 180 deg; joints [33.893, 49.644, 16.689, -143.741, 70.536, -193.734]
  Call Extruder(23151.525)
  MoveL 2445 to (0, 13.33, 105) mm, rotated rx 180 ry 0 rz 180 deg; joints [34.177, 49.357, 17.296, -143.514, 70.861, -193.63]
  Call Extruder(23156.189)
  MoveL 2446 to (-2.97, 13, 105) mm, rotated rx 180 ry 0 rz 180 deg; joints [34.384, 49.025, 17.998, -143.378, 71.207, -193.466]
  Call Extruder(23160.853)
  MoveL 2447 to (-5.78, 12.01, 105) mm, rotated rx 180 ry 0 rz -180 deg; joints [34.5, 48.665, 18.76, -143.34, 71.557, -193.25]
  Call Extruder(23165.516)
  MoveL 2448 to (-8.31, 10.42, 105) mm, rotated rx -180 ry 0 rz -180 deg; joints [34.518, 48.296, 19.544, -143.402, 71.894, -192.995]
  Call Extruder(23170.180)
  MoveL 2449 to (-10.42, 8.31, 105) mm, rotated rx 180 ry 0 rz -180 deg; joints [34.436, 47.937, 20.311, -143.565, 72.202, -192.715]
  Call Extruder(23174.844)
  MoveL 2450 to (-12.01, 5.78, 105) mm, rotated rx 180 ry 0 rz 180 deg; joints [34.254, 47.604, 21.022, -143.822, 72.468, -192.424]
  Call Extruder(23179.508)
  MoveL 2451 to (-13, 2.97, 105) mm, rotated rx -180 ry 0 rz -180 deg; joints [33.981, 47.314, 21.641, -144.163, 72.676, -192.137]
  Call Extruder(23184.172)
  MoveL 2452 to (-13.33, 0, 105) mm, rotated rx 180 ry 0 rz 180 deg; joints [33.63, 47.083, 22.137, -144.571, 72.818, -191.869]
  Call Extruder(23188.835)
  MoveL 2453 to (-12.99, -2.97, 105) mm, rotated rx 180 ry 0 rz -180 deg; joints [33.218, 46.921, 22.484, -145.026, 72.886, -191.632]
  Call Extruder(23193.499)
  MoveL 2454 to (-12.01, -5.78, 105) mm, rotated rx -180 ry 0 rz -180 deg; joints [32.767, 46.837, 22.665, -145.505, 72.875, -191.438]
  Call Extruder(23198.163)
  MoveL 2455 to (-10.42, -8.31, 105) mm, rotated rx 180 ry 0 rz 180 deg; joints [32.302, 46.835, 22.67, -145.982, 72.786, -191.296]
  Call Extruder(23202.827)
  MoveL 2456 to (-8.31, -10.42, 105) mm, rotated rx 180 ry 0 rz -180 deg; joints [31.85, 46.914, 22.499, -146.431, 72.622, -191.211]
  Call Extruder(23207.490)
  MoveL 2457 to (-5.78, -12.01, 105) mm, rotated rx -180 ry 0 rz 180 deg; joints [31.435, 47.072, 22.161, -146.827, 72.39, -191.187]
  Call Extruder(23212.154)
  MoveL 2458 to (-2.97, -12.99, 105) mm, rotated rx -180 ry 0 rz -180 deg; joints [31.079, 47.299, 21.674, -147.148, 72.103, -191.224]
  Call Extruder(23216.818)
  MoveL 2459 to (0, -13.33, 105) mm, rotated rx -180 ry 0 rz -180 deg; joints [30.801, 47.585, 21.061, -147.377, 71.774, -191.321]
  Call Extruder(23221.482)
  MoveL 2460 to (2.97, -12.99, 105) mm, rotated rx 180 ry 0 rz -180 deg; joints [30.614, 47.916, 20.355, -147.503, 71.421, -191.473]
  Set speed (130.0 mm/s)
  MoveL 2461 to (2.97, -12.99, 110) mm, rotated rx 180 ry 0 rz 180 deg; joints [30.614, 47.041, 20.6, -147.387, 70.89, -191.831]
  MoveL 2462 to (-26.25, -4.54, 110) mm, rotated rx 180 ry 0 rz 180 deg; joints [34.172, 44.608, 25.746, -144.214, 73.85, -191.338]
  Call Extruder(23223.715)
  Set speed (60.0 mm/s)
  MoveL 2463 to (-26.09, -5.96, 110) mm, rotated rx 180 ry 0 rz 180 deg; joints [33.969, 44.53, 25.912, -144.436, 73.882, -191.227]
  Call Extruder(23233.079)
  MoveL 2464 to (-24.12, -11.61, 110) mm, rotated rx 180 ry 0 rz 180 deg; joints [33.033, 44.358, 26.28, -145.425, 73.863, -190.844]
  Call Extruder(23242.444)
  MoveL 2465 to (-20.93, -16.69, 110) mm, rotated rx -180 ry 0 rz 180 deg; joints [32.066, 44.353, 26.291, -146.416, 73.688, -190.564]
  Call Extruder(23251.810)
  MoveL 2466 to (-16.69, -20.93, 110) mm, rotated rx -180 ry 0 rz -180 deg; joints [31.126, 44.516, 25.944, -147.35, 73.362, -190.396]
  Call Extruder(23261.174)
  MoveL 2467 to (-11.61, -24.12, 110) mm, rotated rx -180 ry 0 rz 180 deg; joints [30.272, 44.838, 25.258, -148.169, 72.9, -190.344]
  Call Extruder(23270.539)
  MoveL 2468 to (-5.96, -26.09, 110) mm, rotated rx 180 ry 0 rz -180 deg; joints [29.552, 45.303, 24.269, -148.825, 72.324, -190.409]
  Call Extruder(23279.904)
  MoveL 2469 to (0, -26.77, 110) mm, rotated rx 180 ry 0 rz -180 deg; joints [29.003, 45.887, 23.031, -149.283, 71.664, -190.587]
  Call Extruder(23288.195)
  MoveL 2470 to (5.27, -26.17, 110) mm, rotated rx -180 ry 0 rz -180 deg; joints [28.69, 46.484, 21.771, -149.494, 71.035, -190.84]
  Call Extruder(23289.269)
  MoveL 2471 to (5.96, -26.09, 110) mm, rotated rx 180 ry 0 rz 180 deg; joints [28.65, 46.562, 21.606, -149.521, 70.953, -190.873]
  Call Extruder(23298.634)
  MoveL 2472 to (11.61, -24.11, 110) mm, rotated rx 180 ry 0 rz -180 deg; joints [28.503, 47.294, 20.069, -149.53, 70.23, -191.255]
  Call Extruder(23307.999)
  MoveL 2473 to (16.69, -20.93, 110) mm, rotated rx -180 ry 0 rz -180 deg; joints [28.559, 48.046, 18.494, -149.318, 69.533, -191.721]
  Call Extruder(23317.364)
  MoveL 2474 to (20.93, -16.69, 110) mm, rotated rx 180 ry 0 rz 180 deg; joints [28.808, 48.782, 16.961, -148.902, 68.9, -192.251]
  Call Extruder(23326.729)
  MoveL 2475 to (24.12, -11.61, 110) mm, rotated rx -180 ry 0 rz -180 deg; joints [29.229, 49.464, 15.544, -148.311, 68.364, -192.823]
  Call Extruder(23336.094)
  MoveL 2476 to (26.09, -5.96, 110) mm, rotated rx 180 ry 0 rz -180 deg; joints [29.796, 50.058, 14.313, -147.58, 67.954, -193.409]
  Call Extruder(23345.459)
  MoveL 2477 to (26.77, 0, 110) mm, rotated rx -180 ry 0 rz -180 deg; joints [30.482, 50.534, 13.329, -146.749, 67.689, -193.977]
  Call Extruder(23354.824)
  MoveL 2478 to (26.09, 5.96, 110) mm, rotated rx 180 ry 0 rz -180 deg; joints [31.252, 50.868, 12.641, -145.86, 67.584, -194.497]
  Call Extruder(23364.189)
  MoveL 2479 to (24.11, 11.61, 110) mm, rotated rx 180 ry 0 rz -180 deg; joints [32.076, 51.042, 12.282, -144.956, 67.641, -194.939]
  Call Extruder(23373.554)
  MoveL 2480 to (20.93, 16.69, 110) mm, rotated rx 180 ry 0 rz 180 deg; joints [32.917, 51.047, 12.272, -144.077, 67.856, -195.274]
  Call Extruder(23382.919)
  MoveL 2481 to (16.69, 20.93, 110) mm, rotated rx -180 ry 0 rz 180 deg; joints [33.742, 50.883, 12.61, -143.26, 68.215, -195.484]
  Call Extruder(23392.284)
  MoveL 2482 to (11.61, 24.12, 110) mm, rotated rx -180 ry 0 rz -180 deg; joints [34.517, 50.558, 13.28, -142.54, 68.698, -195.555]
  Call Extruder(23401.649)
  MoveL 2483 to (5.96, 26.09, 110) mm, rotated rx 180 ry 0 rz -180 deg; joints [35.208, 50.089, 14.248, -141.944, 69.277, -195.483]
  Call Extruder(23411.014)
  MoveL 2484 to (0, 26.77, 110) mm, rotated rx 180 ry 0 rz 180 deg; joints [35.784, 49.501, 15.466, -141.497, 69.924, -195.273]
  Call Extruder(23420.379)
  MoveL 2485 to (-5.96, 26.09, 110) mm, rotated rx 180 ry 0 rz -180 deg; joints [36.214, 48.824, 16.874, -141.219, 70.607, -194.938]
  Call Extruder(23429.744)
  MoveL 2486 to (-11.61, 24.12, 110) mm, rotated rx 180 ry 0 rz -180 deg; joints [36.473, 48.09, 18.402, -141.126, 71.292, -194.497]
  Call Extruder(23439.109)
  MoveL 2487 to (-16.69, 20.93, 110) mm, rotated rx -180 ry 0 rz -180 deg; joints [36.542, 47.338, 19.976, -141.227, 71.949, -193.976]
  Call Extruder(23448.474)
  MoveL 2488 to (-20.93, 16.69, 110) mm, rotated rx 180 ry 0 rz 180 deg; joints [36.407, 46.604, 21.518, -141.527, 72.548, -193.405]
  Call Extruder(23457.839)
  MoveL 2489 to (-24.12, 11.61, 110) mm, rotated rx -180 ry 0 rz 180 deg; joints [36.065, 45.925, 22.952, -142.019, 73.063, -192.814]
  Call Extruder(23467.204)
  MoveL 2490 to (-26.09, 5.96, 110) mm, rotated rx 180 ry 0 rz 180 deg; joints [35.528, 45.334, 24.203, -142.688, 73.47, -192.235]
  Call Extruder(23476.569)
  MoveL 2491 to (-26.77, 0, 110) mm, rotated rx 180 ry 0 rz 180 deg; joints [34.817, 44.861, 25.207, -143.507, 73.748, -191.697]
  Call Extruder(23481.358)
  MoveL 2492 to (-26.42, -3.05, 110) mm, rotated rx 180 ry 0 rz -180 deg; joints [34.385, 44.69, 25.571, -143.981, 73.816, -191.455]
  Set speed (130.0 mm/s)
  MoveL 2493 to (-41.86, -6.29, 110) mm, rotated rx 180 ry 0 rz 180 deg; joints [35.393, 43.013, 29.168, -143.267, 75.554, -190.546]
  Call Extruder(23486.355)
  Set speed (60.0 mm/s)
  MoveL 2494 to (-41.5, -9.47, 110) mm, rotated rx 180 ry 0 rz 180 deg; joints [34.924, 42.839, 29.544, -143.774, 75.632, -190.304]
  Call Extruder(23501.251)
  MoveL 2495 to (-38.36, -18.47, 110) mm, rotated rx 180 ry 0 rz 180 deg; joints [33.373, 42.564, 30.139, -145.398, 75.623, -189.721]
  Call Extruder(23516.147)
  MoveL 2496 to (-33.29, -26.54, 110) mm, rotated rx -180 ry 0 rz 180 deg; joints [31.763, 42.556, 30.156, -147.039, 75.365, -189.305]
  Call Extruder(23531.043)
  MoveL 2497 to (-26.54, -33.28, 110) mm, rotated rx 180 ry 0 rz -180 deg; joints [30.206, 42.815, 29.594, -148.587, 74.86, -189.062]
  Call Extruder(23545.939)
  MoveL 2498 to (-18.47, -38.36, 110) mm, rotated rx 180 ry 0 rz 180 deg; joints [28.808, 43.329, 28.486, -149.936, 74.13, -188.995]
  Call Extruder(23560.834)
  MoveL 2499 to (-9.47, -41.51, 110) mm, rotated rx -180 ry 0 rz -180 deg; joints [27.654, 44.071, 26.895, -151, 73.209, -189.097]
  Call Extruder(23575.730)
  MoveL 2500 to (0, -42.57, 110) mm, rotated rx 180 ry 0 rz -180 deg; joints [26.805, 45.001, 24.909, -151.721, 72.147, -189.366]
  Call Extruder(23586.786)
  MoveL 2501 to (7.03, -41.78, 110) mm, rotated rx -180 ry 0 rz 180 deg; joints [26.42, 45.796, 23.225, -151.982, 71.298, -189.683]
  Call Extruder(23590.626)
  MoveL 2502 to (9.47, -41.5, 110) mm, rotated rx 180 ry 0 rz -180 deg; joints [26.29, 46.075, 22.633, -152.067, 71.001, -189.793]
  Call Extruder(23605.522)
  MoveL 2503 to (18.47, -38.36, 110) mm, rotated rx 180 ry 0 rz 180 deg; joints [26.114, 47.239, 20.184, -152.037, 69.834, -190.371]
  Call Extruder(23620.418)
  MoveL 2504 to (26.54, -33.28, 110) mm, rotated rx 180 ry 0 rz -180 deg; joints [26.262, 48.436, 17.681, -151.649, 68.71, -191.085]
  Call Extruder(23635.313)
  MoveL 2505 to (33.28, -26.54, 110) mm, rotated rx 180 ry 0 rz 180 deg; joints [26.703, 49.608, 15.246, -150.94, 67.69, -191.912]
  Call Extruder(23650.209)
  MoveL 2506 to (38.36, -18.47, 110) mm, rotated rx 180 ry 0 rz -180 deg; joints [27.4, 50.696, 12.995, -149.961, 66.828, -192.819]
  Call Extruder(23665.105)
  MoveL 2507 to (41.5, -9.47, 110) mm, rotated rx 180 ry 0 rz 180 deg; joints [28.309, 51.647, 11.038, -148.774, 66.171, -193.762]
  Call Extruder(23680.001)
  MoveL 2508 to (42.57, 0, 110) mm, rotated rx 180 ry 0 rz 180 deg; joints [29.382, 52.411, 9.471, -147.445, 65.753, -194.691]
  Call Extruder(23694.897)
  MoveL 2509 to (41.51, 9.47, 110) mm, rotated rx -180 ry 0 rz -180 deg; joints [30.575, 52.947, 8.373, -146.043, 65.595, -195.549]
  Call Extruder(23709.792)
  MoveL 2510 to (38.36, 18.47, 110) mm, rotated rx -180 ry 0 rz 180 deg; joints [31.839, 53.227, 7.801, -144.633, 65.701, -196.282]
  Call Extruder(23724.688)
  MoveL 2511 to (33.28, 26.54, 110) mm, rotated rx 180 ry 0 rz 180 deg; joints [33.128, 53.235, 7.785, -143.277, 66.062, -196.84]
  Call Extruder(23739.584)
  MoveL 2512 to (26.54, 33.29, 110) mm, rotated rx 180 ry 0 rz -180 deg; joints [34.394, 52.971, 8.325, -142.028, 66.652, -197.188]
  Call Extruder(23754.480)
  MoveL 2513 to (18.47, 38.36, 110) mm, rotated rx 180 ry 0 rz 180 deg; joints [35.592, 52.449, 9.393, -140.93, 67.434, -197.303]
  Call Extruder(23769.375)
  MoveL 2514 to (9.47, 41.51, 110) mm, rotated rx 180 ry 0 rz -180 deg; joints [36.675, 51.697, 10.934, -140.019, 68.364, -197.18]
  Call Extruder(23784.271)
  MoveL 2515 to (0, 42.57, 110) mm, rotated rx 180 ry 0 rz -180 deg; joints [37.594, 50.756, 12.871, -139.325, 69.392, -196.829]
  Call Extruder(23799.167)
  MoveL 2516 to (-9.47, 41.5, 110) mm, rotated rx 180 ry 0 rz 180 deg; joints [38.304, 49.675, 15.107, -138.876, 70.467, -196.274]
  Call Extruder(23814.063)
  MoveL 2517 to (-18.47, 38.36, 110) mm, rotated rx -180 ry 0 rz -180 deg; joints [38.762, 48.506, 17.535, -138.696, 71.54, -195.548]
  Call Extruder(23828.959)
  MoveL 2518 to (-26.54, 33.28, 110) mm, rotated rx -180 ry 0 rz -180 deg; joints [38.928, 47.309, 20.037, -138.806, 72.564, -194.695]
  Call Extruder(23843.854)
  MoveL 2519 to (-33.29, 26.54, 110) mm, rotated rx 180 ry 0 rz 180 deg; joints [38.772, 46.142, 22.493, -139.222, 73.499, -193.765]
  Call Extruder(23858.750)
  MoveL 2520 to (-38.36, 18.47, 110) mm, rotated rx 180 ry 0 rz 180 deg; joints [38.277, 45.061, 24.782, -139.95, 74.305, -192.811]
  Call Extruder(23873.646)
  MoveL 2521 to (-41.5, 9.47, 110) mm, rotated rx 180 ry 0 rz -180 deg; joints [37.447, 44.12, 26.788, -140.978, 74.949, -191.884]
  Call Extruder(23888.542)
  MoveL 2522 to (-42.57, 0, 110) mm, rotated rx -180 ry 0 rz 180 deg; joints [36.31, 43.367, 28.405, -142.272, 75.4, -191.035]
  Call Extruder(23896.096)
  MoveL 2523 to (-42.03, -4.8, 110) mm, rotated rx 180 ry 0 rz -180 deg; joints [35.612, 43.095, 28.99, -143.03, 75.518, -190.661]
  Set speed (130.0 mm/s)
  MoveL 2524 to (-54.1, -7.67, 110) mm, rotated rx 180 ry 0 rz -180 deg; joints [36.421, 41.814, 31.768, -142.433, 76.854, -189.923]
  Call Extruder(23900.169)
  Set speed (30.0 mm/s)
  MoveL 2525 to (-53.59, -12.23, 110) mm, rotated rx 180 ry 0 rz -180 deg; joints [35.732, 41.565, 32.312, -143.172, 76.972, -189.582]
  Call Extruder(23911.099)
  MoveL 2526 to (-49.53, -23.85, 110) mm, rotated rx -180 ry 0 rz -180 deg; joints [33.663, 41.208, 33.094, -145.325, 76.985, -188.855]
  Call Extruder(23922.029)
  MoveL 2527 to (-42.98, -34.27, 110) mm, rotated rx 180 ry 0 rz -180 deg; joints [31.506, 41.198, 33.116, -147.517, 76.672, -188.349]
  Call Extruder(23932.959)
  MoveL 2528 to (-34.27, -42.98, 110) mm, rotated rx 180 ry 0 rz 180 deg; joints [29.427, 41.534, 32.378, -149.584, 76.034, -188.065]
  Call Extruder(23943.890)
  MoveL 2529 to (-23.85, -49.53, 110) mm, rotated rx 180 ry 0 rz 180 deg; joints [27.581, 42.2, 30.927, -151.372, 75.092, -187.994]
  Call Extruder(23954.820)
